    |   movel([0.169835, -1.400800, -2.552340, -0.759249, 1.570796, 1.740631],accel_mss,speed_ms,0,blend_radius_m)
    |   movel([0.168721, -1.399189, -2.553525, -0.759676, 1.570796, 1.739517],accel_mss,speed_ms,0,blend_radius_m)
    |   movel([0.167272, -1.397802, -2.554541, -0.760046, 1.570796, 1.738068],accel_mss,speed_ms,0,blend_radius_m)
    |   movel([0.165480, -1.396676, -2.555365, -0.760348, 1.570796, 1.736276],accel_mss,speed_ms,0,blend_radius_m)
    |   movel([0.163342, -1.395840, -2.555975, -0.760574, 1.570796, 1.734139],accel_mss,speed_ms,0,blend_radius_m)
    |   # Splitting Linear movement in 6 (instruction 331: MoveL 300)
    |   movel([0.161964, -1.395450, -2.556260, -0.760680, 1.570796, 1.732760],accel_mss,speed_ms,0,blend_radius_m)
    |   movel([0.160583, -1.395061, -2.556543, -0.760786, 1.570796, 1.731379],accel_mss,speed_ms,0,blend_radius_m)
    |   movel([0.159200, -1.394674, -2.556824, -0.760891, 1.570796, 1.729996],accel_mss,speed_ms,0,blend_radius_m)
    |   movel([0.157815, -1.394290, -2.557104, -0.760996, 1.570796, 1.728611],accel_mss,speed_ms,0,blend_radius_m)
    |   movel([0.156427, -1.393907, -2.557382, -0.761100, 1.570796, 1.727224],accel_mss,speed_ms,0,blend_radius_m)
    |   movel([0.155038, -1.393527, -2.557658, -0.761204, 1.570796, 1.725834],accel_mss,speed_ms,0,blend_radius_m)
    |   # Splitting Linear movement in 18 (instruction 332: MoveL 301)
    |   movel([0.153192, -1.393056, -2.557999, -0.761333, 1.570796, 1.723988],accel_mss,speed_ms,0,blend_radius_m)
    |   movel([0.151342, -1.392590, -2.558337, -0.761462, 1.570796, 1.722138],accel_mss,speed_ms,0,blend_radius_m)
    |   movel([0.149489, -1.392127, -2.558673, -0.761589, 1.570796, 1.720285],accel_mss,speed_ms,0,blend_radius_m)
    |   movel([0.147632, -1.391668, -2.559005, -0.761716, 1.570796, 1.718428],accel_mss,speed_ms,0,blend_radius_m)
    |   movel([0.145771, -1.391213, -2.559334, -0.761842, 1.570796, 1.716568],accel_mss,speed_ms,0,blend_radius_m)
    |   movel([0.143907, -1.390762, -2.559660, -0.761968, 1.570796, 1.714704],accel_mss,speed_ms,0,blend_radius_m)
    |   movel([0.142040, -1.390314, -2.559982, -0.762092, 1.570796, 1.712836],accel_mss,speed_ms,0,blend_radius_m)
    |   movel([0.140169, -1.389871, -2.560302, -0.762216, 1.570796, 1.710965],accel_mss,speed_ms,0,blend_radius_m)
    |   movel([0.138294, -1.389431, -2.560619, -0.762339, 1.570796, 1.709091],accel_mss,speed_ms,0,blend_radius_m)
    |   movel([0.136416, -1.388995, -2.560933, -0.762461, 1.570796, 1.707213],accel_mss,speed_ms,0,blend_radius_m)
    |   movel([0.134535, -1.388563, -2.561243, -0.762583, 1.570796, 1.705331],accel_mss,speed_ms,0,blend_radius_m)
    |   movel([0.132650, -1.388135, -2.561550, -0.762703, 1.570796, 1.703446],accel_mss,speed_ms,0,blend_radius_m)
    |   movel([0.130761, -1.387711, -2.561855, -0.762823, 1.570796, 1.701558],accel_mss,speed_ms,0,blend_radius_m)
    |   movel([0.128869, -1.387291, -2.562156, -0.762942, 1.570796, 1.699666],accel_mss,speed_ms,0,blend_radius_m)
    |   movel([0.126974, -1.386875, -2.562454, -0.763060, 1.570796, 1.697770],accel_mss,speed_ms,0,blend_radius_m)
    |   movel([0.125075, -1.386463, -2.562749, -0.763177, 1.570796, 1.695872],accel_mss,speed_ms,0,blend_radius_m)
    |   movel([0.123173, -1.386055, -2.563041, -0.763293, 1.570796, 1.693969],accel_mss,speed_ms,0,blend_radius_m)
    |   movel([0.121267, -1.385651, -2.563330, -0.763408, 1.570796, 1.692064],accel_mss,speed_ms,0,blend_radius_m)
    |   movel([0.119799, -1.385268, -2.563603, -0.763517, 1.570796, 1.690595],accel_mss,speed_ms,0,blend_radius_m)
    |   movel([0.119411, -1.385044, -2.563763, -0.763581, 1.570796, 1.690207],accel_mss,speed_ms,0,blend_radius_m)
    |   movel([0.119247, -1.384741, -2.563979, -0.763668, 1.570796, 1.690044],accel_mss,speed_ms,0,blend_radius_m)
    |   movel([0.119299, -1.384311, -2.564286, -0.763792, 1.570796, 1.690095],accel_mss,speed_ms,0,blend_radius_m)
    |   movel([0.119560, -1.383712, -2.564713, -0.763964, 1.570796, 1.690357],accel_mss,speed_ms,0,blend_radius_m)
    |   movel([0.120675, -1.381827, -2.566051, -0.764510, 1.570796, 1.691472],accel_mss,speed_ms,0,blend_radius_m)
    |   movel([0.122734, -1.382263, -2.565743, -0.764384, 1.570796, 1.693530],accel_mss,speed_ms,0,blend_radius_m)
    |   speed_ms = 0.005
    |   # Splitting Linear movement in 4 (instruction 341: MoveL 309)
    |   movel([0.122734, -1.380104, -2.564747, -0.767538, 1.570796, 1.693530],accel_mss,speed_ms,0,blend_radius_m)
    |   movel([0.122734, -1.377955, -2.563748, -0.770686, 1.570796, 1.693530],accel_mss,speed_ms,0,blend_radius_m)
    |   movel([0.122734, -1.375816, -2.562745, -0.773828, 1.570796, 1.693530],accel_mss,speed_ms,0,blend_radius_m)
    |   movel([0.122734, -1.373687, -2.561739, -0.776963, 1.570796, 1.693530],accel_mss,speed_ms,0,blend_radius_m)
    |   speed_ms = 0.040
    |   # Splitting Linear movement in 18 (instruction 343: MoveL 310)
    |   movel([0.125073, -1.372444, -2.562608, -0.777337, 1.570796, 1.695869],accel_mss,speed_ms,0,blend_radius_m)
    |   movel([0.127416, -1.371202, -2.563475, -0.777712, 1.570796, 1.698212],accel_mss,speed_ms,0,blend_radius_m)
    |   movel([0.129763, -1.369961, -2.564339, -0.778089, 1.570796, 1.700560],accel_mss,speed_ms,0,blend_radius_m)
    |   movel([0.132116, -1.368721, -2.565200, -0.778468, 1.570796, 1.702912],accel_mss,speed_ms,0,blend_radius_m)
    |   movel([0.134472, -1.367482, -2.566059, -0.778849, 1.570796, 1.705269],accel_mss,speed_ms,0,blend_radius_m)
    |   movel([0.136834, -1.366243, -2.566914, -0.779232, 1.570796, 1.707630],accel_mss,speed_ms,0,blend_radius_m)
    |   movel([0.139200, -1.365006, -2.567767, -0.779616, 1.570796, 1.709996],accel_mss,speed_ms,0,blend_radius_m)
    |   movel([0.141570, -1.363769, -2.568617, -0.780003, 1.570796, 1.712366],accel_mss,speed_ms,0,blend_radius_m)
    |   movel([0.143945, -1.362533, -2.569465, -0.780391, 1.570796, 1.714741],accel_mss,speed_ms,0,blend_radius_m)
    |   movel([0.146324, -1.361298, -2.570309, -0.780781, 1.570796, 1.717121],accel_mss,speed_ms,0,blend_radius_m)
    |   movel([0.148708, -1.360065, -2.571151, -0.781173, 1.570796, 1.719505],accel_mss,speed_ms,0,blend_radius_m)
    |   movel([0.151097, -1.358832, -2.571990, -0.781567, 1.570796, 1.721893],accel_mss,speed_ms,0,blend_radius_m)
    |   movel([0.153490, -1.357600, -2.572826, -0.781962, 1.570796, 1.724286],accel_mss,speed_ms,0,blend_radius_m)
    |   movel([0.155887, -1.356370, -2.573660, -0.782360, 1.570796, 1.726684],accel_mss,speed_ms,0,blend_radius_m)
    |   movel([0.158289, -1.355140, -2.574490, -0.782759, 1.570796, 1.729086],accel_mss,speed_ms,0,blend_radius_m)
    |   movel([0.160696, -1.353911, -2.575318, -0.783159, 1.570796, 1.731492],accel_mss,speed_ms,0,blend_radius_m)
    |   movel([0.163106, -1.352684, -2.576143, -0.783562, 1.570796, 1.733903],accel_mss,speed_ms,0,blend_radius_m)
    |   movel([0.165522, -1.351458, -2.576965, -0.783966, 1.570796, 1.736318],accel_mss,speed_ms,0,blend_radius_m)
    |   speed_ms = 0.005
    |   # Splitting Linear movement in 6 (instruction 345: MoveL 311)
    |   movel([0.165522, -1.352900, -2.577653, -0.781836, 1.570796, 1.736318],accel_mss,speed_ms,0,blend_radius_m)
    |   movel([0.165522, -1.354347, -2.578339, -0.779703, 1.570796, 1.736318],accel_mss,speed_ms,0,blend_radius_m)
    |   movel([0.165522, -1.355799, -2.579023, -0.777567, 1.570796, 1.736318],accel_mss,speed_ms,0,blend_radius_m)
    |   movel([0.165522, -1.357255, -2.579705, -0.775428, 1.570796, 1.736318],accel_mss,speed_ms,0,blend_radius_m)
    |   movel([0.165522, -1.358716, -2.580386, -0.773287, 1.570796, 1.736318],accel_mss,speed_ms,0,blend_radius_m)
    |   movel([0.165522, -1.360182, -2.581065, -0.771142, 1.570796, 1.736318],accel_mss,speed_ms,0,blend_radius_m)
    |   speed_ms = 0.035
    |   movel([0.167244, -1.360441, -2.580889, -0.771058, 1.570796, 1.738040],accel_mss,speed_ms,0,blend_radius_m)
    |   movel([0.168585, -1.360439, -2.580891, -0.771059, 1.570796, 1.739382],accel_mss,speed_ms,0,blend_radius_m)
    |   movel([0.169955, -1.360315, -2.580975, -0.771099, 1.570796, 1.740751],accel_mss,speed_ms,0,blend_radius_m)
    |   movel([0.171344, -1.360075, -2.581138, -0.771176, 1.570796, 1.742141],accel_mss,speed_ms,0,blend_radius_m)
    |   movel([0.172746, -1.359724, -2.581376, -0.771289, 1.570796, 1.743542],accel_mss,speed_ms,0,blend_radius_m)
    |   movel([0.174155, -1.359265, -2.581687, -0.771437, 1.570796, 1.744951],accel_mss,speed_ms,0,blend_radius_m)
    |   movel([0.176950, -1.358045, -2.582512, -0.771832, 1.570796, 1.747746],accel_mss,speed_ms,0,blend_radius_m)
    |   movel([0.178323, -1.357292, -2.583020, -0.772077, 1.570796, 1.749120],accel_mss,speed_ms,0,blend_radius_m)
    |   movel([0.180981, -1.355525, -2.584210, -0.772655, 1.570796, 1.751777],accel_mss,speed_ms,0,blend_radius_m)
    |   movel([0.182252, -1.354517, -2.584886, -0.772986, 1.570796, 1.753048],accel_mss,speed_ms,0,blend_radius_m)
    |   movel([0.184624, -1.352283, -2.586380, -0.773726, 1.570796, 1.755420],accel_mss,speed_ms,0,blend_radius_m)
    |   movel([0.185715, -1.351062, -2.587194, -0.774133, 1.570796, 1.756511],accel_mss,speed_ms,0,blend_radius_m)
    |   movel([0.186729, -1.349776, -2.588049, -0.774564, 1.570796, 1.757525],accel_mss,speed_ms,0,blend_radius_m)
    |   movel([0.187656, -1.348435, -2.588938, -0.775016, 1.570796, 1.758453],accel_mss,speed_ms,0,blend_radius_m)
    |   movel([0.188445, -1.347113, -2.589812, -0.775464, 1.570796, 1.759241],accel_mss,speed_ms,0,blend_radius_m)
    |   movel([0.189111, -1.345791, -2.590684, -0.775914, 1.570796, 1.759907],accel_mss,speed_ms,0,blend_radius_m)
    |   movel([0.190069, -1.343183, -2.592397, -0.776810, 1.570796, 1.760866],accel_mss,speed_ms,0,blend_radius_m)
    |   movel([0.190366, -1.341908, -2.593230, -0.777251, 1.570796, 1.761162],accel_mss,speed_ms,0,blend_radius_m)
    |   movel([0.190585, -1.339465, -2.594822, -0.778102, 1.570796, 1.761381],accel_mss,speed_ms,0,blend_radius_m)
    |   movel([0.190509, -1.338309, -2.595572, -0.778508, 1.570796, 1.761306],accel_mss,speed_ms,0,blend_radius_m)
    |   movel([0.189997, -1.336168, -2.596957, -0.779265, 1.570796, 1.760793],accel_mss,speed_ms,0,blend_radius_m)
    |   movel([0.189557, -1.335195, -2.597584, -0.779610, 1.570796, 1.760353],accel_mss,speed_ms,0,blend_radius_m)
    |   movel([0.188317, -1.333493, -2.598678, -0.780218, 1.570796, 1.759113],accel_mss,speed_ms,0,blend_radius_m)
    |   movel([0.187516, -1.332779, -2.599136, -0.780474, 1.570796, 1.758312],accel_mss,speed_ms,0,blend_radius_m)
    |   movel([0.186599, -1.332164, -2.599530, -0.780696, 1.570796, 1.757395],accel_mss,speed_ms,0,blend_radius_m)
    |   movel([0.185562, -1.331657, -2.599854, -0.780878, 1.570796, 1.756358],accel_mss,speed_ms,0,blend_radius_m)
    |   movel([0.183890, -1.331154, -2.600175, -0.781060, 1.570796, 1.754686],accel_mss,speed_ms,0,blend_radius_m)
    |   movel([0.183257, -1.331163, -2.600169, -0.781057, 1.570796, 1.754053],accel_mss,speed_ms,0,blend_radius_m)
    |   movel([0.182728, -1.331365, -2.600040, -0.780983, 1.570796, 1.753524],accel_mss,speed_ms,0,blend_radius_m)
    |   movel([0.182274, -1.331780, -2.599775, -0.780834, 1.570796, 1.753070],accel_mss,speed_ms,0,blend_radius_m)
    |   movel([0.181874, -1.332416, -2.599368, -0.780605, 1.570796, 1.752671],accel_mss,speed_ms,0,blend_radius_m)
    |   movel([0.181131, -1.334429, -2.598077, -0.779883, 1.570796, 1.751927],accel_mss,speed_ms,0,blend_radius_m)
    |   movel([0.182746, -1.334997, -2.597711, -0.779681, 1.570796, 1.753542],accel_mss,speed_ms,0,blend_radius_m)
    |   movel([0.184246, -1.335833, -2.597173, -0.779383, 1.570796, 1.755043],accel_mss,speed_ms,0,blend_radius_m)
    |   movel([0.185396, -1.336953, -2.596450, -0.778986, 1.570796, 1.756192],accel_mss,speed_ms,0,blend_radius_m)
    |   movel([0.186193, -1.338317, -2.595567, -0.778505, 1.570796, 1.756989],accel_mss,speed_ms,0,blend_radius_m)
    |   movel([0.186629, -1.339885, -2.594549, -0.777955, 1.570796, 1.757425],accel_mss,speed_ms,0,blend_radius_m)
    |   movel([0.186702, -1.341619, -2.593419, -0.777351, 1.570796, 1.757498],accel_mss,speed_ms,0,blend_radius_m)
    |   movel([0.186412, -1.343480, -2.592202, -0.776707, 1.570796, 1.757208],accel_mss,speed_ms,0,blend_radius_m)
    |   movel([0.185753, -1.345430, -2.590921, -0.776037, 1.570796, 1.756550],accel_mss,speed_ms,0,blend_radius_m)
    |   movel([0.184722, -1.347430, -2.589603, -0.775356, 1.570796, 1.755519],accel_mss,speed_ms,0,blend_radius_m)
    |   movel([0.183346, -1.349406, -2.588295, -0.774688, 1.570796, 1.754142],accel_mss,speed_ms,0,blend_radius_m)
    |   movel([0.181729, -1.351210, -2.587095, -0.774083, 1.570796, 1.752525],accel_mss,speed_ms,0,blend_radius_m)
    |   movel([0.179917, -1.352823, -2.586020, -0.773546, 1.570796, 1.750714],accel_mss,speed_ms,0,blend_radius_m)
    |   movel([0.177958, -1.354214, -2.585089, -0.773086, 1.570796, 1.748754],accel_mss,speed_ms,0,blend_radius_m)
    |   movel([0.175895, -1.355355, -2.584323, -0.772710, 1.570796, 1.746691],accel_mss,speed_ms,0,blend_radius_m)
    |   movel([0.173775, -1.356220, -2.583742, -0.772427, 1.570796, 1.744572],accel_mss,speed_ms,0,blend_radius_m)
    |   movel([0.171644, -1.356782, -2.583364, -0.772243, 1.570796, 1.742441],accel_mss,speed_ms,0,blend_radius_m)
    |   movel([0.169547, -1.357011, -2.583210, -0.772169, 1.570796, 1.740343],accel_mss,speed_ms,0,blend_radius_m)
    |   movel([0.167897, -1.357114, -2.583140, -0.772135, 1.570796, 1.738693],accel_mss,speed_ms,0,blend_radius_m)
    |   movel([0.167339, -1.357255, -2.583045, -0.772089, 1.570796, 1.738135],accel_mss,speed_ms,0,blend_radius_m)
    |   movel([0.166903, -1.357499, -2.582881, -0.772010, 1.570796, 1.737699],accel_mss,speed_ms,0,blend_radius_m)
    |   movel([0.166548, -1.357878, -2.582625, -0.771886, 1.570796, 1.737344],accel_mss,speed_ms,0,blend_radius_m)
    |   movel([0.166226, -1.358432, -2.582251, -0.771707, 1.570796, 1.737022],accel_mss,speed_ms,0,blend_radius_m)
    |   movel([0.165522, -1.360182, -2.581065, -0.771142, 1.570796, 1.736318],accel_mss,speed_ms,0,blend_radius_m)
    |   movel([0.167244, -1.360441, -2.580889, -0.771058, 1.570796, 1.738040],accel_mss,speed_ms,0,blend_radius_m)
    |   movel([0.167727, -1.360442, -2.580889, -0.771058, 1.570796, 1.738523],accel_mss,speed_ms,0,blend_radius_m)
    |   speed_ms = 0.005
    |   # Splitting Linear movement in 6 (instruction 405: MoveL 369)
    |   movel([0.167727, -1.358977, -2.580210, -0.773202, 1.570796, 1.738523],accel_mss,speed_ms,0,blend_radius_m)
    |   movel([0.167727, -1.357516, -2.579529, -0.775344, 1.570796, 1.738523],accel_mss,speed_ms,0,blend_radius_m)
    |   movel([0.167727, -1.356060, -2.578847, -0.777482, 1.570796, 1.738523],accel_mss,speed_ms,0,blend_radius_m)
    |   movel([0.167727, -1.354609, -2.578163, -0.779618, 1.570796, 1.738523],accel_mss,speed_ms,0,blend_radius_m)
    |   movel([0.167727, -1.353162, -2.577477, -0.781750, 1.570796, 1.738523],accel_mss,speed_ms,0,blend_radius_m)
    |   movel([0.167727, -1.351720, -2.576790, -0.783879, 1.570796, 1.738523],accel_mss,speed_ms,0,blend_radius_m)
    |   speed_ms = 0.040
    |   # Splitting Linear movement in 6 (instruction 407: MoveL 370)
    |   movel([0.165743, -1.351292, -2.577077, -0.784021, 1.570796, 1.736539],accel_mss,speed_ms,0,blend_radius_m)
    |   movel([0.163755, -1.350868, -2.577360, -0.784161, 1.570796, 1.734551],accel_mss,speed_ms,0,blend_radius_m)
    |   movel([0.161764, -1.350449, -2.577640, -0.784300, 1.570796, 1.732560],accel_mss,speed_ms,0,blend_radius_m)
    |   movel([0.159768, -1.350034, -2.577917, -0.784438, 1.570796, 1.730565],accel_mss,speed_ms,0,blend_radius_m)
    |   movel([0.157769, -1.349624, -2.578191, -0.784574, 1.570796, 1.728566],accel_mss,speed_ms,0,blend_radius_m)
    |   movel([0.155767, -1.349218, -2.578462, -0.784709, 1.570796, 1.726563],accel_mss,speed_ms,0,blend_radius_m)
    |   speed_ms = 0.005
    |   # Splitting Linear movement in 6 (instruction 409: MoveL 371)
    |   movel([0.155767, -1.350663, -2.579151, -0.782575, 1.570796, 1.726563],accel_mss,speed_ms,0,blend_radius_m)
    |   movel([0.155767, -1.352112, -2.579838, -0.780439, 1.570796, 1.726563],accel_mss,speed_ms,0,blend_radius_m)
    |   movel([0.155767, -1.353567, -2.580524, -0.778299, 1.570796, 1.726563],accel_mss,speed_ms,0,blend_radius_m)
    |   movel([0.155767, -1.355025, -2.581208, -0.776156, 1.570796, 1.726563],accel_mss,speed_ms,0,blend_radius_m)
    |   movel([0.155767, -1.356489, -2.581891, -0.774010, 1.570796, 1.726563],accel_mss,speed_ms,0,blend_radius_m)
    |   movel([0.155767, -1.357957, -2.582571, -0.771861, 1.570796, 1.726563],accel_mss,speed_ms,0,blend_radius_m)
    |   speed_ms = 0.035
    |   movel([0.157355, -1.355183, -2.584439, -0.772767, 1.570796, 1.728151],accel_mss,speed_ms,0,blend_radius_m)
    |   movel([0.158736, -1.352483, -2.586247, -0.773659, 1.570796, 1.729532],accel_mss,speed_ms,0,blend_radius_m)
    |   movel([0.159906, -1.349859, -2.587994, -0.774536, 1.570796, 1.730702],accel_mss,speed_ms,0,blend_radius_m)
    |   movel([0.160863, -1.347310, -2.589682, -0.775397, 1.570796, 1.731660],accel_mss,speed_ms,0,blend_radius_m)
    |   movel([0.161608, -1.344839, -2.591310, -0.776240, 1.570796, 1.732405],accel_mss,speed_ms,0,blend_radius_m)
    |   movel([0.162137, -1.342441, -2.592882, -0.777066, 1.570796, 1.732933],accel_mss,speed_ms,0,blend_radius_m)
    |   movel([0.162447, -1.340121, -2.594395, -0.777873, 1.570796, 1.733244],accel_mss,speed_ms,0,blend_radius_m)
    |   movel([0.162537, -1.337882, -2.595848, -0.778658, 1.570796, 1.733334],accel_mss,speed_ms,0,blend_radius_m)
    |   movel([0.162403, -1.335721, -2.597245, -0.779423, 1.570796, 1.733200],accel_mss,speed_ms,0,blend_radius_m)
    |   movel([0.162046, -1.333638, -2.598585, -0.780166, 1.570796, 1.732842],accel_mss,speed_ms,0,blend_radius_m)
    |   movel([0.161461, -1.331638, -2.599866, -0.780885, 1.570796, 1.732257],accel_mss,speed_ms,0,blend_radius_m)
    |   movel([0.160647, -1.329720, -2.601089, -0.781580, 1.570796, 1.731443],accel_mss,speed_ms,0,blend_radius_m)
    |   movel([0.159603, -1.327887, -2.602254, -0.782248, 1.570796, 1.730399],accel_mss,speed_ms,0,blend_radius_m)
    |   movel([0.158326, -1.326137, -2.603362, -0.782890, 1.570796, 1.729123],accel_mss,speed_ms,0,blend_radius_m)
    |   movel([0.156817, -1.324475, -2.604410, -0.783504, 1.570796, 1.727613],accel_mss,speed_ms,0,blend_radius_m)
    |   movel([0.155070, -1.322901, -2.605399, -0.784089, 1.570796, 1.725866],accel_mss,speed_ms,0,blend_radius_m)
    |   movel([0.156422, -1.321887, -2.606034, -0.784467, 1.570796, 1.727219],accel_mss,speed_ms,0,blend_radius_m)
    |   movel([0.158344, -1.320258, -2.607053, -0.785078, 1.570796, 1.729140],accel_mss,speed_ms,0,blend_radius_m)
    |   movel([0.160279, -1.321620, -2.606202, -0.784567, 1.570796, 1.731076],accel_mss,speed_ms,0,blend_radius_m)
    |   movel([0.161946, -1.323240, -2.605186, -0.783963, 1.570796, 1.732742],accel_mss,speed_ms,0,blend_radius_m)
    |   movel([0.163339, -1.325091, -2.604022, -0.783276, 1.570796, 1.734136],accel_mss,speed_ms,0,blend_radius_m)
    |   movel([0.164467, -1.327149, -2.602721, -0.782518, 1.570796, 1.735263],accel_mss,speed_ms,0,blend_radius_m)
    |   movel([0.165329, -1.329385, -2.601302, -0.781701, 1.570796, 1.736126],accel_mss,speed_ms,0,blend_radius_m)
    |   movel([0.165930, -1.331777, -2.599777, -0.780835, 1.570796, 1.736726],accel_mss,speed_ms,0,blend_radius_m)
    |   movel([0.166274, -1.334295, -2.598163, -0.779931, 1.570796, 1.737070],accel_mss,speed_ms,0,blend_radius_m)
    |   movel([0.166364, -1.336915, -2.596474, -0.779000, 1.570796, 1.737160],accel_mss,speed_ms,0,blend_radius_m)
    |   movel([0.166202, -1.339614, -2.594725, -0.778050, 1.570796, 1.736998],accel_mss,speed_ms,0,blend_radius_m)
    |   movel([0.165795, -1.342364, -2.592932, -0.777093, 1.570796, 1.736591],accel_mss,speed_ms,0,blend_radius_m)
    |   movel([0.165144, -1.345146, -2.591108, -0.776135, 1.570796, 1.735940],accel_mss,speed_ms,0,blend_radius_m)
    |   movel([0.164254, -1.347930, -2.589272, -0.775187, 1.570796, 1.735050],accel_mss,speed_ms,0,blend_radius_m)
    |   movel([0.163128, -1.350701, -2.587435, -0.774254, 1.570796, 1.733924],accel_mss,speed_ms,0,blend_radius_m)
    |   movel([0.161769, -1.353431, -2.585613, -0.773345, 1.570796, 1.732566],accel_mss,speed_ms,0,blend_radius_m)
    |   movel([0.160179, -1.356100, -2.583823, -0.772466, 1.570796, 1.730976],accel_mss,speed_ms,0,blend_radius_m)
    |   movel([0.158366, -1.358687, -2.582078, -0.771624, 1.570796, 1.729162],accel_mss,speed_ms,0,blend_radius_m)
    |   movel([0.155767, -1.357957, -2.582571, -0.771861, 1.570796, 1.726563],accel_mss,speed_ms,0,blend_radius_m)
    |   movel([0.157104, -1.355619, -2.584147, -0.772624, 1.570796, 1.727901],accel_mss,speed_ms,0,blend_radius_m)
    |   speed_ms = 0.005
    |   # Splitting Linear movement in 6 (instruction 448: MoveL 408)
    |   movel([0.157104, -1.354148, -2.583464, -0.774777, 1.570796, 1.727901],accel_mss,speed_ms,0,blend_radius_m)
    |   movel([0.157104, -1.352682, -2.582780, -0.776927, 1.570796, 1.727901],accel_mss,speed_ms,0,blend_radius_m)
    |   movel([0.157104, -1.351221, -2.582094, -0.779075, 1.570796, 1.727901],accel_mss,speed_ms,0,blend_radius_m)
    |   movel([0.157104, -1.349764, -2.581406, -0.781219, 1.570796, 1.727901],accel_mss,speed_ms,0,blend_radius_m)
    |   movel([0.157104, -1.348312, -2.580717, -0.783360, 1.570796, 1.727901],accel_mss,speed_ms,0,blend_radius_m)
    |   movel([0.157104, -1.346865, -2.580026, -0.785498, 1.570796, 1.727901],accel_mss,speed_ms,0,blend_radius_m)
    |   speed_ms = 0.040
    |   # Splitting Linear movement in 6 (instruction 450: MoveL 409)
    |   movel([0.154683, -1.347404, -2.579668, -0.785317, 1.570796, 1.725480],accel_mss,speed_ms,0,blend_radius_m)
    |   movel([0.152263, -1.347947, -2.579307, -0.785134, 1.570796, 1.723059],accel_mss,speed_ms,0,blend_radius_m)
    |   movel([0.149843, -1.348495, -2.578943, -0.784951, 1.570796, 1.720639],accel_mss,speed_ms,0,blend_radius_m)
    |   movel([0.147424, -1.349048, -2.578575, -0.784766, 1.570796, 1.718220],accel_mss,speed_ms,0,blend_radius_m)
    |   movel([0.145005, -1.349604, -2.578204, -0.784581, 1.570796, 1.715801],accel_mss,speed_ms,0,blend_radius_m)
    |   movel([0.142587, -1.350165, -2.577830, -0.784394, 1.570796, 1.713383],accel_mss,speed_ms,0,blend_radius_m)
    |   speed_ms = 0.005
    |   # Splitting Linear movement in 6 (instruction 452: MoveL 410)
    |   movel([0.142587, -1.351609, -2.578518, -0.782262, 1.570796, 1.713383],accel_mss,speed_ms,0,blend_radius_m)
    |   movel([0.142587, -1.353057, -2.579205, -0.780127, 1.570796, 1.713383],accel_mss,speed_ms,0,blend_radius_m)
    |   movel([0.142587, -1.354510, -2.579890, -0.777989, 1.570796, 1.713383],accel_mss,speed_ms,0,blend_radius_m)
    |   movel([0.142587, -1.355968, -2.580574, -0.775847, 1.570796, 1.713383],accel_mss,speed_ms,0,blend_radius_m)
    |   movel([0.142587, -1.357430, -2.581256, -0.773703, 1.570796, 1.713383],accel_mss,speed_ms,0,blend_radius_m)
    |   movel([0.142587, -1.358897, -2.581936, -0.771556, 1.570796, 1.713383],accel_mss,speed_ms,0,blend_radius_m)
    |   speed_ms = 0.035
    |   movel([0.144618, -1.357853, -2.582642, -0.771895, 1.570796, 1.715414],accel_mss,speed_ms,0,blend_radius_m)
    |   movel([0.145265, -1.357609, -2.582806, -0.771974, 1.570796, 1.716061],accel_mss,speed_ms,0,blend_radius_m)
    |   movel([0.145714, -1.357563, -2.582837, -0.771989, 1.570796, 1.716510],accel_mss,speed_ms,0,blend_radius_m)
    |   movel([0.146013, -1.357716, -2.582734, -0.771939, 1.570796, 1.716810],accel_mss,speed_ms,0,blend_radius_m)
    |   movel([0.146199, -1.358079, -2.582489, -0.771821, 1.570796, 1.716996],accel_mss,speed_ms,0,blend_radius_m)
    |   movel([0.146391, -1.359451, -2.581561, -0.771377, 1.570796, 1.717188],accel_mss,speed_ms,0,blend_radius_m)
    |   movel([0.146678, -1.361399, -2.580239, -0.770751, 1.570796, 1.717475],accel_mss,speed_ms,0,blend_radius_m)
    |   movel([0.147186, -1.363219, -2.578999, -0.770171, 1.570796, 1.717982],accel_mss,speed_ms,0,blend_radius_m)
    |   movel([0.147904, -1.364903, -2.577847, -0.769639, 1.570796, 1.718700],accel_mss,speed_ms,0,blend_radius_m)
    |   movel([0.148823, -1.366444, -2.576790, -0.769155, 1.570796, 1.719620],accel_mss,speed_ms,0,blend_radius_m)
    |   movel([0.149928, -1.367838, -2.575830, -0.768720, 1.570796, 1.720724],accel_mss,speed_ms,0,blend_radius_m)
    |   movel([0.151213, -1.369078, -2.574975, -0.768336, 1.570796, 1.722009],accel_mss,speed_ms,0,blend_radius_m)
    |   movel([0.152668, -1.370158, -2.574228, -0.768003, 1.570796, 1.723464],accel_mss,speed_ms,0,blend_radius_m)
    |   movel([0.154279, -1.371073, -2.573594, -0.767722, 1.570796, 1.725075],accel_mss,speed_ms,0,blend_radius_m)
    |   movel([0.156039, -1.371815, -2.573079, -0.767495, 1.570796, 1.726835],accel_mss,speed_ms,0,blend_radius_m)
    |   movel([0.157942, -1.372376, -2.572689, -0.767324, 1.570796, 1.728738],accel_mss,speed_ms,0,blend_radius_m)
    |   movel([0.159972, -1.372753, -2.572427, -0.767209, 1.570796, 1.730769],accel_mss,speed_ms,0,blend_radius_m)
    |   movel([0.162127, -1.372933, -2.572301, -0.767155, 1.570796, 1.732924],accel_mss,speed_ms,0,blend_radius_m)
    |   movel([0.164395, -1.372914, -2.572314, -0.767160, 1.570796, 1.735192],accel_mss,speed_ms,0,blend_radius_m)
    |   movel([0.166771, -1.372686, -2.572473, -0.767230, 1.570796, 1.737567],accel_mss,speed_ms,0,blend_radius_m)
    |   movel([0.169243, -1.372241, -2.572783, -0.767365, 1.570796, 1.740039],accel_mss,speed_ms,0,blend_radius_m)
    |   movel([0.171807, -1.371570, -2.573249, -0.767570, 1.570796, 1.742603],accel_mss,speed_ms,0,blend_radius_m)
    |   movel([0.174557, -1.370640, -2.573894, -0.767855, 1.570796, 1.745353],accel_mss,speed_ms,0,blend_radius_m)
    |   movel([0.177244, -1.369534, -2.574660, -0.768195, 1.570796, 1.748040],accel_mss,speed_ms,0,blend_radius_m)
    |   movel([0.179860, -1.368264, -2.575537, -0.768588, 1.570796, 1.750657],accel_mss,speed_ms,0,blend_radius_m)
    |   movel([0.182392, -1.366838, -2.576519, -0.769032, 1.570796, 1.753189],accel_mss,speed_ms,0,blend_radius_m)
    |   movel([0.184834, -1.365264, -2.577600, -0.769525, 1.570796, 1.755630],accel_mss,speed_ms,0,blend_radius_m)
    |   movel([0.187171, -1.363557, -2.578768, -0.770064, 1.570796, 1.757967],accel_mss,speed_ms,0,blend_radius_m)
    |   movel([0.189395, -1.361724, -2.580018, -0.770647, 1.570796, 1.760191],accel_mss,speed_ms,0,blend_radius_m)
    |   movel([0.191497, -1.359772, -2.581343, -0.771274, 1.570796, 1.762293],accel_mss,speed_ms,0,blend_radius_m)
    |   movel([0.193462, -1.357715, -2.582735, -0.771939, 1.570796, 1.764258],accel_mss,speed_ms,0,blend_radius_m)
    |   movel([0.195284, -1.355561, -2.584185, -0.772643, 1.570796, 1.766080],accel_mss,speed_ms,0,blend_radius_m)
    |   movel([0.196947, -1.353323, -2.585686, -0.773381, 1.570796, 1.767743],accel_mss,speed_ms,0,blend_radius_m)
    |   movel([0.198441, -1.351008, -2.587230, -0.774151, 1.570796, 1.769238],accel_mss,speed_ms,0,blend_radius_m)
    |   movel([0.199751, -1.348631, -2.588808, -0.774950, 1.570796, 1.770547],accel_mss,speed_ms,0,blend_radius_m)
    |   movel([0.200870, -1.346200, -2.590415, -0.775775, 1.570796, 1.771666],accel_mss,speed_ms,0,blend_radius_m)
    |   movel([0.201780, -1.343726, -2.592041, -0.776623, 1.570796, 1.772576],accel_mss,speed_ms,0,blend_radius_m)
    |   movel([0.202469, -1.341224, -2.593677, -0.777488, 1.570796, 1.773266],accel_mss,speed_ms,0,blend_radius_m)
    |   movel([0.202849, -1.339180, -2.595007, -0.778202, 1.570796, 1.773645],accel_mss,speed_ms,0,blend_radius_m)
    |   movel([0.203044, -1.337202, -2.596289, -0.778898, 1.570796, 1.773841],accel_mss,speed_ms,0,blend_radius_m)
    |   movel([0.203058, -1.335296, -2.597519, -0.779574, 1.570796, 1.773854],accel_mss,speed_ms,0,blend_radius_m)
    |   movel([0.202894, -1.333475, -2.598690, -0.780225, 1.570796, 1.773690],accel_mss,speed_ms,0,blend_radius_m)
    |   movel([0.202553, -1.331740, -2.599801, -0.780848, 1.570796, 1.773349],accel_mss,speed_ms,0,blend_radius_m)
    |   movel([0.202041, -1.330104, -2.600845, -0.781440, 1.570796, 1.772837],accel_mss,speed_ms,0,blend_radius_m)
    |   movel([0.201360, -1.328572, -2.601819, -0.781998, 1.570796, 1.772156],accel_mss,speed_ms,0,blend_radius_m)
    |   movel([0.200513, -1.327155, -2.602718, -0.782516, 1.570796, 1.771309],accel_mss,speed_ms,0,blend_radius_m)
    |   movel([0.199505, -1.325856, -2.603539, -0.782994, 1.570796, 1.770301],accel_mss,speed_ms,0,blend_radius_m)
    |   movel([0.198339, -1.324688, -2.604276, -0.783425, 1.570796, 1.769136],accel_mss,speed_ms,0,blend_radius_m)
    |   movel([0.197021, -1.323655, -2.604925, -0.783808, 1.570796, 1.767817],accel_mss,speed_ms,0,blend_radius_m)
    |   movel([0.195555, -1.322767, -2.605483, -0.784139, 1.570796, 1.766352],accel_mss,speed_ms,0,blend_radius_m)
    |   movel([0.193946, -1.322030, -2.605945, -0.784414, 1.570796, 1.764742],accel_mss,speed_ms,0,blend_radius_m)
    |   movel([0.192197, -1.321452, -2.606307, -0.784630, 1.570796, 1.762993],accel_mss,speed_ms,0,blend_radius_m)
    |   movel([0.190314, -1.321041, -2.606564, -0.784784, 1.570796, 1.761110],accel_mss,speed_ms,0,blend_radius_m)
    |   movel([0.188302, -1.320804, -2.606712, -0.784873, 1.570796, 1.759098],accel_mss,speed_ms,0,blend_radius_m)
    |   movel([0.186033, -1.320586, -2.606848, -0.784955, 1.570796, 1.756829],accel_mss,speed_ms,0,blend_radius_m)
    |   movel([0.186699, -1.318620, -2.608073, -0.785696, 1.570796, 1.757495],accel_mss,speed_ms,0,blend_radius_m)
    |   movel([0.187062, -1.317970, -2.608477, -0.785942, 1.570796, 1.757858],accel_mss,speed_ms,0,blend_radius_m)
    |   movel([0.187486, -1.317514, -2.608760, -0.786115, 1.570796, 1.758283],accel_mss,speed_ms,0,blend_radius_m)
    |   movel([0.188004, -1.317220, -2.608942, -0.786227, 1.570796, 1.758800],accel_mss,speed_ms,0,blend_radius_m)
    |   movel([0.188643, -1.317067, -2.609037, -0.786285, 1.570796, 1.759439],accel_mss,speed_ms,0,blend_radius_m)
    |   movel([0.190414, -1.317087, -2.609024, -0.786277, 1.570796, 1.761210],accel_mss,speed_ms,0,blend_radius_m)
    |   movel([0.192754, -1.317403, -2.608829, -0.786157, 1.570796, 1.763550],accel_mss,speed_ms,0,blend_radius_m)
    |   movel([0.194935, -1.317924, -2.608505, -0.785960, 1.570796, 1.765732],accel_mss,speed_ms,0,blend_radius_m)
    |   movel([0.196955, -1.318641, -2.608060, -0.785688, 1.570796, 1.767752],accel_mss,speed_ms,0,blend_radius_m)
    |   movel([0.198804, -1.319549, -2.607495, -0.785345, 1.570796, 1.769600],accel_mss,speed_ms,0,blend_radius_m)
    |   movel([0.200476, -1.320635, -2.606817, -0.784936, 1.570796, 1.771272],accel_mss,speed_ms,0,blend_radius_m)
    |   movel([0.201971, -1.321889, -2.606033, -0.784467, 1.570796, 1.772767],accel_mss,speed_ms,0,blend_radius_m)
    |   movel([0.203277, -1.323305, -2.605146, -0.783939, 1.570796, 1.774073],accel_mss,speed_ms,0,blend_radius_m)
    |   movel([0.204395, -1.324866, -2.604164, -0.783359, 1.570796, 1.775192],accel_mss,speed_ms,0,blend_radius_m)
    |   movel([0.205318, -1.326569, -2.603089, -0.782731, 1.570796, 1.776115],accel_mss,speed_ms,0,blend_radius_m)
    |   movel([0.206044, -1.328398, -2.601930, -0.782061, 1.570796, 1.776841],accel_mss,speed_ms,0,blend_radius_m)
    |   movel([0.206568, -1.330347, -2.600690, -0.781352, 1.570796, 1.777365],accel_mss,speed_ms,0,blend_radius_m)
    |   movel([0.206883, -1.332405, -2.599375, -0.780609, 1.570796, 1.777680],accel_mss,speed_ms,0,blend_radius_m)
    |   movel([0.206991, -1.334560, -2.597992, -0.779836, 1.570796, 1.777788],accel_mss,speed_ms,0,blend_radius_m)
    |   movel([0.206884, -1.336808, -2.596543, -0.779038, 1.570796, 1.777681],accel_mss,speed_ms,0,blend_radius_m)
    |   movel([0.206563, -1.339132, -2.595038, -0.778219, 1.570796, 1.777359],accel_mss,speed_ms,0,blend_radius_m)
    |   movel([0.206022, -1.341527, -2.593479, -0.777383, 1.570796, 1.776818],accel_mss,speed_ms,0,blend_radius_m)
    |   movel([0.205270, -1.343944, -2.591898, -0.776547, 1.570796, 1.776066],accel_mss,speed_ms,0,blend_radius_m)
    |   movel([0.204329, -1.346344, -2.590319, -0.775725, 1.570796, 1.775125],accel_mss,speed_ms,0,blend_radius_m)
    |   movel([0.203206, -1.348721, -2.588749, -0.774919, 1.570796, 1.774003],accel_mss,speed_ms,0,blend_radius_m)
    |   movel([0.201915, -1.351058, -2.587197, -0.774134, 1.570796, 1.772711],accel_mss,speed_ms,0,blend_radius_m)
    |   movel([0.200464, -1.353349, -2.585668, -0.773372, 1.570796, 1.771260],accel_mss,speed_ms,0,blend_radius_m)
    |   movel([0.198867, -1.355583, -2.584170, -0.772635, 1.570796, 1.769664],accel_mss,speed_ms,0,blend_radius_m)
    |   movel([0.197131, -1.357754, -2.582708, -0.771926, 1.570796, 1.767927],accel_mss,speed_ms,0,blend_radius_m)
    |   movel([0.195269, -1.359848, -2.581292, -0.771249, 1.570796, 1.766065],accel_mss,speed_ms,0,blend_radius_m)
    |   movel([0.193289, -1.361860, -2.579925, -0.770604, 1.570796, 1.764085],accel_mss,speed_ms,0,blend_radius_m)
    |   movel([0.191199, -1.363780, -2.578616, -0.769993, 1.570796, 1.761995],accel_mss,speed_ms,0,blend_radius_m)
    |   movel([0.189008, -1.365597, -2.577371, -0.769420, 1.570796, 1.759805],accel_mss,speed_ms,0,blend_radius_m)
    |   movel([0.186730, -1.367307, -2.576197, -0.768886, 1.570796, 1.757527],accel_mss,speed_ms,0,blend_radius_m)
    |   movel([0.184369, -1.368895, -2.575102, -0.768393, 1.570796, 1.755166],accel_mss,speed_ms,0,blend_radius_m)
    |   movel([0.181935, -1.370360, -2.574089, -0.767941, 1.570796, 1.752731],accel_mss,speed_ms,0,blend_radius_m)
    |   movel([0.179436, -1.371687, -2.573168, -0.767534, 1.570796, 1.750233],accel_mss,speed_ms,0,blend_radius_m)
    |   movel([0.176882, -1.372869, -2.572346, -0.767174, 1.570796, 1.747678],accel_mss,speed_ms,0,blend_radius_m)
    |   movel([0.174330, -1.373880, -2.571641, -0.766868, 1.570796, 1.745127],accel_mss,speed_ms,0,blend_radius_m)
    |   movel([0.171808, -1.374709, -2.571062, -0.766618, 1.570796, 1.742604],accel_mss,speed_ms,0,blend_radius_m)
    |   movel([0.169325, -1.375362, -2.570606, -0.766421, 1.570796, 1.740121],accel_mss,speed_ms,0,blend_radius_m)
    |   movel([0.166894, -1.375835, -2.570275, -0.766280, 1.570796, 1.737691],accel_mss,speed_ms,0,blend_radius_m)
    |   movel([0.164518, -1.376135, -2.570065, -0.766190, 1.570796, 1.735315],accel_mss,speed_ms,0,blend_radius_m)
    |   movel([0.162212, -1.376262, -2.569975, -0.766152, 1.570796, 1.733009],accel_mss,speed_ms,0,blend_radius_m)
    |   movel([0.159981, -1.376220, -2.570004, -0.766164, 1.570796, 1.730778],accel_mss,speed_ms,0,blend_radius_m)
    |   movel([0.157837, -1.376006, -2.570155, -0.766228, 1.570796, 1.728633],accel_mss,speed_ms,0,blend_radius_m)
    |   movel([0.155786, -1.375625, -2.570421, -0.766342, 1.570796, 1.726582],accel_mss,speed_ms,0,blend_radius_m)
    |   movel([0.153843, -1.375077, -2.570805, -0.766507, 1.570796, 1.724639],accel_mss,speed_ms,0,blend_radius_m)
    |   movel([0.152016, -1.374360, -2.571306, -0.766723, 1.570796, 1.722813],accel_mss,speed_ms,0,blend_radius_m)
    |   movel([0.150314, -1.373478, -2.571922, -0.766990, 1.570796, 1.721111],accel_mss,speed_ms,0,blend_radius_m)
    |   movel([0.148748, -1.372430, -2.572651, -0.767308, 1.570796, 1.719545],accel_mss,speed_ms,0,blend_radius_m)
    |   movel([0.147329, -1.371214, -2.573496, -0.767679, 1.570796, 1.718125],accel_mss,speed_ms,0,blend_radius_m)
    |   movel([0.146068, -1.369834, -2.574453, -0.768103, 1.570796, 1.716865],accel_mss,speed_ms,0,blend_radius_m)
    |   movel([0.144973, -1.368285, -2.575522, -0.768581, 1.570796, 1.715770],accel_mss,speed_ms,0,blend_radius_m)
    |   movel([0.143879, -1.366214, -2.576948, -0.769227, 1.570796, 1.714675],accel_mss,speed_ms,0,blend_radius_m)
    |   movel([0.143082, -1.363974, -2.578483, -0.769932, 1.570796, 1.713878],accel_mss,speed_ms,0,blend_radius_m)
    |   movel([0.142634, -1.361542, -2.580141, -0.770705, 1.570796, 1.713430],accel_mss,speed_ms,0,blend_radius_m)
    |   movel([0.142587, -1.358897, -2.581936, -0.771556, 1.570796, 1.713383],accel_mss,speed_ms,0,blend_radius_m)
    |   movel([0.144618, -1.357853, -2.582642, -0.771895, 1.570796, 1.715414],accel_mss,speed_ms,0,blend_radius_m)
    |   movel([0.145130, -1.357660, -2.582771, -0.771957, 1.570796, 1.715926],accel_mss,speed_ms,0,blend_radius_m)
    |   speed_ms = 0.005
    |   # Splitting Linear movement in 4 (instruction 570: MoveL 526)
    |   movel([0.145130, -1.355460, -2.581749, -0.775180, 1.570796, 1.715926],accel_mss,speed_ms,0,blend_radius_m)
    |   movel([0.145130, -1.353269, -2.580723, -0.778397, 1.570796, 1.715926],accel_mss,speed_ms,0,blend_radius_m)
    |   movel([0.145130, -1.351089, -2.579694, -0.781606, 1.570796, 1.715926],accel_mss,speed_ms,0,blend_radius_m)
    |   movel([0.145130, -1.348920, -2.578660, -0.784809, 1.570796, 1.715926],accel_mss,speed_ms,0,blend_radius_m)
    |   speed_ms = 0.040
    |   # Splitting Linear movement in 10 (instruction 572: MoveL 527)
    |   movel([0.142834, -1.349486, -2.578283, -0.784620, 1.570796, 1.713630],accel_mss,speed_ms,0,blend_radius_m)
    |   movel([0.140539, -1.350055, -2.577903, -0.784431, 1.570796, 1.711335],accel_mss,speed_ms,0,blend_radius_m)
    |   movel([0.138244, -1.350629, -2.577520, -0.784240, 1.570796, 1.709040],accel_mss,speed_ms,0,blend_radius_m)
    |   movel([0.135951, -1.351206, -2.577134, -0.784049, 1.570796, 1.706747],accel_mss,speed_ms,0,blend_radius_m)
    |   movel([0.133658, -1.351786, -2.576745, -0.783857, 1.570796, 1.704454],accel_mss,speed_ms,0,blend_radius_m)
    |   movel([0.131366, -1.352370, -2.576354, -0.783665, 1.570796, 1.702162],accel_mss,speed_ms,0,blend_radius_m)
    |   movel([0.129075, -1.352958, -2.575959, -0.783472, 1.570796, 1.699871],accel_mss,speed_ms,0,blend_radius_m)
    |   movel([0.126784, -1.353549, -2.575562, -0.783278, 1.570796, 1.697581],accel_mss,speed_ms,0,blend_radius_m)
    |   movel([0.124495, -1.354144, -2.575161, -0.783083, 1.570796, 1.695291],accel_mss,speed_ms,0,blend_radius_m)
    |   movel([0.122207, -1.354743, -2.574758, -0.782888, 1.570796, 1.693003],accel_mss,speed_ms,0,blend_radius_m)
    |   speed_ms = 0.005
    |   # Splitting Linear movement in 4 (instruction 574: MoveL 528)
    |   movel([0.122207, -1.356903, -2.575785, -0.779701, 1.570796, 1.693003],accel_mss,speed_ms,0,blend_radius_m)
    |   movel([0.122207, -1.359074, -2.576808, -0.776507, 1.570796, 1.693003],accel_mss,speed_ms,0,blend_radius_m)
    |   movel([0.122207, -1.361255, -2.577828, -0.773306, 1.570796, 1.693003],accel_mss,speed_ms,0,blend_radius_m)
    |   movel([0.122207, -1.363446, -2.578844, -0.770099, 1.570796, 1.693003],accel_mss,speed_ms,0,blend_radius_m)
    |   speed_ms = 0.035
    |   movel([0.120628, -1.366409, -2.576814, -0.769166, 1.570796, 1.691424],accel_mss,speed_ms,0,blend_radius_m)
    |   movel([0.119214, -1.366251, -2.576922, -0.769215, 1.570796, 1.690010],accel_mss,speed_ms,0,blend_radius_m)
    |   movel([0.117940, -1.365961, -2.577122, -0.769306, 1.570796, 1.688737],accel_mss,speed_ms,0,blend_radius_m)
    |   movel([0.116802, -1.365543, -2.577409, -0.769438, 1.570796, 1.687599],accel_mss,speed_ms,0,blend_radius_m)
    |   movel([0.115794, -1.365001, -2.577780, -0.769608, 1.570796, 1.686590],accel_mss,speed_ms,0,blend_radius_m)
    |   movel([0.114907, -1.364338, -2.578234, -0.769817, 1.570796, 1.685704],accel_mss,speed_ms,0,blend_radius_m)
    |   movel([0.114139, -1.363559, -2.578767, -0.770064, 1.570796, 1.684935],accel_mss,speed_ms,0,blend_radius_m)
    |   movel([0.113482, -1.362670, -2.579373, -0.770346, 1.570796, 1.684278],accel_mss,speed_ms,0,blend_radius_m)
    |   movel([0.112927, -1.361672, -2.580053, -0.770664, 1.570796, 1.683724],accel_mss,speed_ms,0,blend_radius_m)
    |   movel([0.112291, -1.359794, -2.581329, -0.771267, 1.570796, 1.683087],accel_mss,speed_ms,0,blend_radius_m)
    |   movel([0.112068, -1.357735, -2.582721, -0.771933, 1.570796, 1.682864],accel_mss,speed_ms,0,blend_radius_m)
    |   movel([0.112247, -1.355538, -2.584201, -0.772650, 1.570796, 1.683043],accel_mss,speed_ms,0,blend_radius_m)
    |   movel([0.112813, -1.353248, -2.585735, -0.773405, 1.570796, 1.683610],accel_mss,speed_ms,0,blend_radius_m)
    |   movel([0.113756, -1.350904, -2.587299, -0.774186, 1.570796, 1.684553],accel_mss,speed_ms,0,blend_radius_m)
    |   movel([0.115059, -1.348556, -2.588858, -0.774975, 1.570796, 1.685855],accel_mss,speed_ms,0,blend_radius_m)
    |   movel([0.116712, -1.346243, -2.590386, -0.775760, 1.570796, 1.687508],accel_mss,speed_ms,0,blend_radius_m)
    |   movel([0.118694, -1.344015, -2.591851, -0.776523, 1.570796, 1.689491],accel_mss,speed_ms,0,blend_radius_m)
    |   movel([0.120927, -1.341975, -2.593187, -0.777228, 1.570796, 1.691723],accel_mss,speed_ms,0,blend_radius_m)
    |   movel([0.123311, -1.340195, -2.594347, -0.777847, 1.570796, 1.694107],accel_mss,speed_ms,0,blend_radius_m)
    |   movel([0.125806, -1.338693, -2.595323, -0.778373, 1.570796, 1.696602],accel_mss,speed_ms,0,blend_radius_m)
    |   movel([0.128360, -1.337495, -2.596099, -0.778795, 1.570796, 1.699157],accel_mss,speed_ms,0,blend_radius_m)
    |   movel([0.130924, -1.336621, -2.596664, -0.779104, 1.570796, 1.701720],accel_mss,speed_ms,0,blend_radius_m)
    |   movel([0.133454, -1.336091, -2.597007, -0.779292, 1.570796, 1.704250],accel_mss,speed_ms,0,blend_radius_m)
    |   movel([0.135896, -1.335925, -2.597114, -0.779351, 1.570796, 1.706692],accel_mss,speed_ms,0,blend_radius_m)
    |   movel([0.138205, -1.336142, -2.596974, -0.779274, 1.570796, 1.709002],accel_mss,speed_ms,0,blend_radius_m)
    |   movel([0.140282, -1.336752, -2.596579, -0.779057, 1.570796, 1.711078],accel_mss,speed_ms,0,blend_radius_m)
    |   movel([0.142032, -1.337718, -2.595955, -0.778716, 1.570796, 1.712829],accel_mss,speed_ms,0,blend_radius_m)
    |   movel([0.143439, -1.339008, -2.595118, -0.778262, 1.570796, 1.714235],accel_mss,speed_ms,0,blend_radius_m)
    |   movel([0.144488, -1.340588, -2.594091, -0.777710, 1.570796, 1.715284],accel_mss,speed_ms,0,blend_radius_m)
    |   movel([0.145165, -1.342423, -2.592894, -0.777072, 1.570796, 1.715961],accel_mss,speed_ms,0,blend_radius_m)
    |   movel([0.145455, -1.344478, -2.591547, -0.776364, 1.570796, 1.716251],accel_mss,speed_ms,0,blend_radius_m)
    |   movel([0.145344, -1.346722, -2.590071, -0.775597, 1.570796, 1.716141],accel_mss,speed_ms,0,blend_radius_m)
    |   movel([0.144824, -1.349115, -2.588487, -0.774786, 1.570796, 1.715620],accel_mss,speed_ms,0,blend_radius_m)
    |   movel([0.144168, -1.350936, -2.587278, -0.774175, 1.570796, 1.714964],accel_mss,speed_ms,0,blend_radius_m)
    |   movel([0.143799, -1.351553, -2.586867, -0.773969, 1.570796, 1.714595],accel_mss,speed_ms,0,blend_radius_m)
    |   movel([0.143353, -1.352016, -2.586559, -0.773815, 1.570796, 1.714149],accel_mss,speed_ms,0,blend_radius_m)
    |   movel([0.142793, -1.352352, -2.586334, -0.773703, 1.570796, 1.713589],accel_mss,speed_ms,0,blend_radius_m)
    |   movel([0.142084, -1.352591, -2.586175, -0.773623, 1.570796, 1.712880],accel_mss,speed_ms,0,blend_radius_m)
    |   movel([0.140076, -1.352892, -2.585973, -0.773523, 1.570796, 1.710872],accel_mss,speed_ms,0,blend_radius_m)
    |   movel([0.140788, -1.349617, -2.588155, -0.774617, 1.570796, 1.711585],accel_mss,speed_ms,0,blend_radius_m)
    |   movel([0.141097, -1.346826, -2.590002, -0.775561, 1.570796, 1.711893],accel_mss,speed_ms,0,blend_radius_m)
    |   movel([0.140994, -1.344508, -2.591528, -0.776354, 1.570796, 1.711790],accel_mss,speed_ms,0,blend_radius_m)
    |   movel([0.140462, -1.342652, -2.592744, -0.776993, 1.570796, 1.711258],accel_mss,speed_ms,0,blend_radius_m)
    |   movel([0.140033, -1.341891, -2.593241, -0.777256, 1.570796, 1.710829],accel_mss,speed_ms,0,blend_radius_m)
    |   movel([0.139494, -1.341240, -2.593666, -0.777483, 1.570796, 1.710290],accel_mss,speed_ms,0,blend_radius_m)
    |   movel([0.138842, -1.340698, -2.594020, -0.777671, 1.570796, 1.709638],accel_mss,speed_ms,0,blend_radius_m)
    |   movel([0.137202, -1.339931, -2.594519, -0.777939, 1.570796, 1.707998],accel_mss,speed_ms,0,blend_radius_m)
    |   movel([0.136209, -1.339702, -2.594668, -0.778019, 1.570796, 1.707005],accel_mss,speed_ms,0,blend_radius_m)
    |   movel([0.133874, -1.339543, -2.594771, -0.778075, 1.570796, 1.704670],accel_mss,speed_ms,0,blend_radius_m)
    |   movel([0.131737, -1.339758, -2.594631, -0.778000, 1.570796, 1.702534],accel_mss,speed_ms,0,blend_radius_m)
    |   movel([0.129547, -1.340326, -2.594262, -0.777801, 1.570796, 1.700343],accel_mss,speed_ms,0,blend_radius_m)
    |   movel([0.127354, -1.341213, -2.593684, -0.777492, 1.570796, 1.698150],accel_mss,speed_ms,0,blend_radius_m)
    |   movel([0.125210, -1.342385, -2.592919, -0.777086, 1.570796, 1.696007],accel_mss,speed_ms,0,blend_radius_m)
    |   movel([0.123173, -1.343809, -2.591986, -0.776594, 1.570796, 1.693969],accel_mss,speed_ms,0,blend_radius_m)
    |   movel([0.121287, -1.345453, -2.590906, -0.776030, 1.570796, 1.692083],accel_mss,speed_ms,0,blend_radius_m)
    |   movel([0.119605, -1.347280, -2.589702, -0.775407, 1.570796, 1.690401],accel_mss,speed_ms,0,blend_radius_m)
    |   movel([0.118176, -1.349262, -2.588390, -0.774737, 1.570796, 1.688972],accel_mss,speed_ms,0,blend_radius_m)
    |   movel([0.116876, -1.351632, -2.586814, -0.773942, 1.570796, 1.687673],accel_mss,speed_ms,0,blend_radius_m)
    |   movel([0.116086, -1.353795, -2.585370, -0.773224, 1.570796, 1.686883],accel_mss,speed_ms,0,blend_radius_m)
    |   movel([0.115884, -1.354803, -2.584694, -0.772892, 1.570796, 1.686680],accel_mss,speed_ms,0,blend_radius_m)
    |   movel([0.115866, -1.356690, -2.583426, -0.772273, 1.570796, 1.686662],accel_mss,speed_ms,0,blend_radius_m)
    |   movel([0.116049, -1.357571, -2.582832, -0.771986, 1.570796, 1.686846],accel_mss,speed_ms,0,blend_radius_m)
    |   movel([0.116806, -1.359220, -2.581717, -0.771452, 1.570796, 1.687602],accel_mss,speed_ms,0,blend_radius_m)
    |   movel([0.118084, -1.360738, -2.580688, -0.770963, 1.570796, 1.688880],accel_mss,speed_ms,0,blend_radius_m)
    |   movel([0.119883, -1.362140, -2.579735, -0.770515, 1.570796, 1.690680],accel_mss,speed_ms,0,blend_radius_m)
    |   movel([0.122207, -1.363446, -2.578844, -0.770099, 1.570796, 1.693003],accel_mss,speed_ms,0,blend_radius_m)
    |   movel([0.120970, -1.365764, -2.577257, -0.769368, 1.570796, 1.691767],accel_mss,speed_ms,0,blend_radius_m)
    |   speed_ms = 0.005
    |   # Splitting Linear movement in 4 (instruction 644: MoveL 596)
    |   movel([0.120970, -1.363576, -2.576244, -0.772569, 1.570796, 1.691767],accel_mss,speed_ms,0,blend_radius_m)
    |   movel([0.120970, -1.361399, -2.575227, -0.775763, 1.570796, 1.691767],accel_mss,speed_ms,0,blend_radius_m)
    |   movel([0.120970, -1.359233, -2.574206, -0.778950, 1.570796, 1.691767],accel_mss,speed_ms,0,blend_radius_m)
    |   movel([0.120970, -1.357076, -2.573181, -0.782131, 1.570796, 1.691767],accel_mss,speed_ms,0,blend_radius_m)
    |   speed_ms = 0.040
    |   # Splitting Linear movement in 18 (instruction 646: MoveL 597)
    |   movel([0.120281, -1.355463, -2.574272, -0.782653, 1.570796, 1.691078],accel_mss,speed_ms,0,blend_radius_m)
    |   movel([0.119589, -1.353848, -2.575361, -0.783180, 1.570796, 1.690386],accel_mss,speed_ms,0,blend_radius_m)
    |   movel([0.118894, -1.352231, -2.576448, -0.783711, 1.570796, 1.689691],accel_mss,speed_ms,0,blend_radius_m)
    |   movel([0.118196, -1.350611, -2.577532, -0.784246, 1.570796, 1.688993],accel_mss,speed_ms,0,blend_radius_m)
    |   movel([0.117496, -1.348989, -2.578614, -0.784786, 1.570796, 1.688292],accel_mss,speed_ms,0,blend_radius_m)
    |   movel([0.116792, -1.347365, -2.579694, -0.785330, 1.570796, 1.687588],accel_mss,speed_ms,0,blend_radius_m)
    |   movel([0.116085, -1.345739, -2.580772, -0.785878, 1.570796, 1.686882],accel_mss,speed_ms,0,blend_radius_m)
    |   movel([0.115376, -1.344111, -2.581848, -0.786430, 1.570796, 1.686172],accel_mss,speed_ms,0,blend_radius_m)
    |   movel([0.114663, -1.342481, -2.582921, -0.786987, 1.570796, 1.685460],accel_mss,speed_ms,0,blend_radius_m)
    |   movel([0.113948, -1.340849, -2.583992, -0.787548, 1.570796, 1.684744],accel_mss,speed_ms,0,blend_radius_m)
    |   movel([0.113229, -1.339214, -2.585061, -0.788114, 1.570796, 1.684025],accel_mss,speed_ms,0,blend_radius_m)
    |   movel([0.112508, -1.337577, -2.586128, -0.788684, 1.570796, 1.683304],accel_mss,speed_ms,0,blend_radius_m)
    |   movel([0.111783, -1.335939, -2.587193, -0.789258, 1.570796, 1.682579],accel_mss,speed_ms,0,blend_radius_m)
    |   movel([0.111055, -1.334298, -2.588255, -0.789836, 1.570796, 1.681852],accel_mss,speed_ms,0,blend_radius_m)
    |   movel([0.110324, -1.332654, -2.589315, -0.790419, 1.570796, 1.681121],accel_mss,speed_ms,0,blend_radius_m)
    |   movel([0.109590, -1.331009, -2.590373, -0.791007, 1.570796, 1.680387],accel_mss,speed_ms,0,blend_radius_m)
    |   movel([0.108853, -1.329362, -2.591428, -0.791599, 1.570796, 1.679650],accel_mss,speed_ms,0,blend_radius_m)
    |   movel([0.108113, -1.327712, -2.592482, -0.792195, 1.570796, 1.678910],accel_mss,speed_ms,0,blend_radius_m)
    |   speed_ms = 0.005
    |   # Splitting Linear movement in 4 (instruction 648: MoveL 598)
    |   movel([0.108113, -1.329914, -2.593538, -0.788936, 1.570796, 1.678910],accel_mss,speed_ms,0,blend_radius_m)
    |   movel([0.108113, -1.332127, -2.594591, -0.785670, 1.570796, 1.678910],accel_mss,speed_ms,0,blend_radius_m)
    |   movel([0.108113, -1.334352, -2.595641, -0.782397, 1.570796, 1.678910],accel_mss,speed_ms,0,blend_radius_m)
    |   movel([0.108113, -1.336587, -2.596686, -0.779116, 1.570796, 1.678910],accel_mss,speed_ms,0,blend_radius_m)
    |   speed_ms = 0.035
    |   movel([0.106316, -1.338548, -2.595417, -0.778424, 1.570796, 1.677112],accel_mss,speed_ms,0,blend_radius_m)
    |   movel([0.104661, -1.340518, -2.594137, -0.777734, 1.570796, 1.675458],accel_mss,speed_ms,0,blend_radius_m)
    |   movel([0.103151, -1.342493, -2.592848, -0.777048, 1.570796, 1.673947],accel_mss,speed_ms,0,blend_radius_m)
    |   movel([0.101779, -1.344469, -2.591553, -0.776367, 1.570796, 1.672575],accel_mss,speed_ms,0,blend_radius_m)
    |   movel([0.100547, -1.346438, -2.590257, -0.775693, 1.570796, 1.671344],accel_mss,speed_ms,0,blend_radius_m)
    |   movel([0.099454, -1.348400, -2.588962, -0.775028, 1.570796, 1.670250],accel_mss,speed_ms,0,blend_radius_m)
    |   movel([0.098494, -1.350345, -2.587671, -0.774373, 1.570796, 1.669290],accel_mss,speed_ms,0,blend_radius_m)
    |   movel([0.097668, -1.352272, -2.586388, -0.773729, 1.570796, 1.668464],accel_mss,speed_ms,0,blend_radius_m)
    |   movel([0.096975, -1.354174, -2.585116, -0.773099, 1.570796, 1.667771],accel_mss,speed_ms,0,blend_radius_m)
    |   movel([0.096414, -1.356048, -2.583858, -0.772483, 1.570796, 1.667210],accel_mss,speed_ms,0,blend_radius_m)
    |   movel([0.095669, -1.359690, -2.581399, -0.771300, 1.570796, 1.666466],accel_mss,speed_ms,0,blend_radius_m)
    |   movel([0.095485, -1.361452, -2.580203, -0.770734, 1.570796, 1.666281],accel_mss,speed_ms,0,blend_radius_m)
    |   movel([0.095485, -1.364830, -2.577897, -0.769662, 1.570796, 1.666281],accel_mss,speed_ms,0,blend_radius_m)
    |   movel([0.095663, -1.366440, -2.576793, -0.769156, 1.570796, 1.666459],accel_mss,speed_ms,0,blend_radius_m)
    |   movel([0.096371, -1.369483, -2.574695, -0.768211, 1.570796, 1.667167],accel_mss,speed_ms,0,blend_radius_m)
    |   movel([0.096895, -1.370908, -2.573708, -0.767773, 1.570796, 1.667692],accel_mss,speed_ms,0,blend_radius_m)
    |   movel([0.098286, -1.373539, -2.571879, -0.766971, 1.570796, 1.669082],accel_mss,speed_ms,0,blend_radius_m)
    |   movel([0.099145, -1.374741, -2.571040, -0.766608, 1.570796, 1.669941],accel_mss,speed_ms,0,blend_radius_m)
    |   movel([0.101187, -1.376891, -2.569534, -0.765964, 1.570796, 1.671984],accel_mss,speed_ms,0,blend_radius_m)
    |   movel([0.102370, -1.377834, -2.568871, -0.765684, 1.570796, 1.673166],accel_mss,speed_ms,0,blend_radius_m)
    |   movel([0.103656, -1.378683, -2.568274, -0.765432, 1.570796, 1.674453],accel_mss,speed_ms,0,blend_radius_m)
    |   movel([0.105046, -1.379436, -2.567743, -0.765210, 1.570796, 1.675842],accel_mss,speed_ms,0,blend_radius_m)
    |   movel([0.106539, -1.380083, -2.567286, -0.765020, 1.570796, 1.677335],accel_mss,speed_ms,0,blend_radius_m)
    |   movel([0.108133, -1.380628, -2.566901, -0.764860, 1.570796, 1.678929],accel_mss,speed_ms,0,blend_radius_m)
    |   movel([0.109829, -1.381061, -2.566595, -0.764734, 1.570796, 1.680626],accel_mss,speed_ms,0,blend_radius_m)
    |   movel([0.111627, -1.381379, -2.566369, -0.764641, 1.570796, 1.682423],accel_mss,speed_ms,0,blend_radius_m)
    |   movel([0.113523, -1.381580, -2.566227, -0.764582, 1.570796, 1.684320],accel_mss,speed_ms,0,blend_radius_m)
    |   movel([0.112735, -1.383387, -2.564944, -0.764058, 1.570796, 1.683531],accel_mss,speed_ms,0,blend_radius_m)
    |   movel([0.112369, -1.384047, -2.564474, -0.763868, 1.570796, 1.683166],accel_mss,speed_ms,0,blend_radius_m)
    |   movel([0.111916, -1.384464, -2.564177, -0.763748, 1.570796, 1.682713],accel_mss,speed_ms,0,blend_radius_m)
    |   movel([0.111348, -1.384668, -2.564032, -0.763689, 1.570796, 1.682144],accel_mss,speed_ms,0,blend_radius_m)
    |   movel([0.110638, -1.384685, -2.564020, -0.763685, 1.570796, 1.681434],accel_mss,speed_ms,0,blend_radius_m)
    |   movel([0.107947, -1.384329, -2.564273, -0.763787, 1.570796, 1.678743],accel_mss,speed_ms,0,blend_radius_m)
    |   movel([0.105434, -1.383717, -2.564709, -0.763963, 1.570796, 1.676230],accel_mss,speed_ms,0,blend_radius_m)
    |   movel([0.103104, -1.382861, -2.565318, -0.764210, 1.570796, 1.673901],accel_mss,speed_ms,0,blend_radius_m)
    |   movel([0.100967, -1.381773, -2.566090, -0.764526, 1.570796, 1.671763],accel_mss,speed_ms,0,blend_radius_m)
    |   movel([0.099025, -1.380467, -2.567014, -0.764907, 1.570796, 1.669822],accel_mss,speed_ms,0,blend_radius_m)
    |   movel([0.097291, -1.378954, -2.568083, -0.765352, 1.570796, 1.668087],accel_mss,speed_ms,0,blend_radius_m)
    |   movel([0.095771, -1.377246, -2.569285, -0.765858, 1.570796, 1.666568],accel_mss,speed_ms,0,blend_radius_m)
    |   movel([0.094473, -1.375356, -2.570610, -0.766423, 1.570796, 1.665270],accel_mss,speed_ms,0,blend_radius_m)
    |   movel([0.093411, -1.373293, -2.572051, -0.767046, 1.570796, 1.664208],accel_mss,speed_ms,0,blend_radius_m)
    |   movel([0.092590, -1.371070, -2.573596, -0.767723, 1.570796, 1.663386],accel_mss,speed_ms,0,blend_radius_m)
    |   movel([0.092021, -1.368697, -2.575238, -0.768454, 1.570796, 1.662818],accel_mss,speed_ms,0,blend_radius_m)
    |   movel([0.091719, -1.366186, -2.576967, -0.769236, 1.570796, 1.662515],accel_mss,speed_ms,0,blend_radius_m)
    |   movel([0.091688, -1.363552, -2.578771, -0.770066, 1.570796, 1.662485],accel_mss,speed_ms,0,blend_radius_m)
    |   movel([0.091943, -1.360805, -2.580642, -0.770941, 1.570796, 1.662739],accel_mss,speed_ms,0,blend_radius_m)
    |   movel([0.092496, -1.357956, -2.582572, -0.771861, 1.570796, 1.663292],accel_mss,speed_ms,0,blend_radius_m)
    |   movel([0.093354, -1.355018, -2.584550, -0.772821, 1.570796, 1.664150],accel_mss,speed_ms,0,blend_radius_m)
    |   movel([0.095047, -1.350740, -2.587409, -0.774241, 1.570796, 1.665843],accel_mss,speed_ms,0,blend_radius_m)
    |   movel([0.096067, -1.348618, -2.588817, -0.774954, 1.570796, 1.666864],accel_mss,speed_ms,0,blend_radius_m)
    |   movel([0.097206, -1.346508, -2.590212, -0.775670, 1.570796, 1.668002],accel_mss,speed_ms,0,blend_radius_m)
    |   movel([0.098471, -1.344407, -2.591594, -0.776388, 1.570796, 1.669267],accel_mss,speed_ms,0,blend_radius_m)
    |   movel([0.099865, -1.342317, -2.592963, -0.777109, 1.570796, 1.670662],accel_mss,speed_ms,0,blend_radius_m)
    |   movel([0.101395, -1.340234, -2.594321, -0.777833, 1.570796, 1.672192],accel_mss,speed_ms,0,blend_radius_m)
    |   movel([0.103062, -1.338162, -2.595667, -0.778560, 1.570796, 1.673858],accel_mss,speed_ms,0,blend_radius_m)
    |   movel([0.104534, -1.336491, -2.596748, -0.779150, 1.570796, 1.675330],accel_mss,speed_ms,0,blend_radius_m)
    |   movel([0.105082, -1.336014, -2.597056, -0.779319, 1.570796, 1.675878],accel_mss,speed_ms,0,blend_radius_m)
    |   movel([0.105579, -1.335755, -2.597223, -0.779411, 1.570796, 1.676375],accel_mss,speed_ms,0,blend_radius_m)
    |   movel([0.106077, -1.335699, -2.597259, -0.779431, 1.570796, 1.676873],accel_mss,speed_ms,0,blend_radius_m)
    |   movel([0.106628, -1.335829, -2.597175, -0.779385, 1.570796, 1.677424],accel_mss,speed_ms,0,blend_radius_m)
    |   movel([0.108113, -1.336587, -2.596686, -0.779116, 1.570796, 1.678910],accel_mss,speed_ms,0,blend_radius_m)
    |   movel([0.106316, -1.338548, -2.595417, -0.778424, 1.570796, 1.677112],accel_mss,speed_ms,0,blend_radius_m)
    |   movel([0.106109, -1.338793, -2.595258, -0.778338, 1.570796, 1.676906],accel_mss,speed_ms,0,blend_radius_m)
    |   speed_ms = 0.005
    |   # Splitting Linear movement in 6 (instruction 714: MoveL 662)
    |   movel([0.106109, -1.337304, -2.594563, -0.780522, 1.570796, 1.676906],accel_mss,speed_ms,0,blend_radius_m)
    |   movel([0.106109, -1.335819, -2.593867, -0.782703, 1.570796, 1.676906],accel_mss,speed_ms,0,blend_radius_m)
    |   movel([0.106109, -1.334340, -2.593168, -0.784880, 1.570796, 1.676906],accel_mss,speed_ms,0,blend_radius_m)
    |   movel([0.106109, -1.332866, -2.592468, -0.787055, 1.570796, 1.676906],accel_mss,speed_ms,0,blend_radius_m)
    |   movel([0.106109, -1.331396, -2.591767, -0.789226, 1.570796, 1.676906],accel_mss,speed_ms,0,blend_radius_m)
    |   movel([0.106109, -1.329932, -2.591064, -0.791393, 1.570796, 1.676906],accel_mss,speed_ms,0,blend_radius_m)
    |   speed_ms = 0.040
    |   # Splitting Linear movement in 20 (instruction 716: MoveL 663)
    |   movel([0.106875, -1.327668, -2.592510, -0.792211, 1.570796, 1.677671],accel_mss,speed_ms,0,blend_radius_m)
    |   movel([0.107644, -1.325396, -2.593955, -0.793038, 1.570796, 1.678441],accel_mss,speed_ms,0,blend_radius_m)
    |   movel([0.108418, -1.323116, -2.595398, -0.793875, 1.570796, 1.679214],accel_mss,speed_ms,0,blend_radius_m)
    |   movel([0.109195, -1.320828, -2.596839, -0.794722, 1.570796, 1.679991],accel_mss,speed_ms,0,blend_radius_m)
    |   movel([0.109976, -1.318531, -2.598279, -0.795579, 1.570796, 1.680773],accel_mss,speed_ms,0,blend_radius_m)
    |   movel([0.110761, -1.316226, -2.599717, -0.796446, 1.570796, 1.681558],accel_mss,speed_ms,0,blend_radius_m)
    |   movel([0.111551, -1.313912, -2.601153, -0.797324, 1.570796, 1.682347],accel_mss,speed_ms,0,blend_radius_m)
    |   movel([0.112344, -1.311590, -2.602588, -0.798212, 1.570796, 1.683140],accel_mss,speed_ms,0,blend_radius_m)
    |   movel([0.113141, -1.309259, -2.604021, -0.799110, 1.570796, 1.683938],accel_mss,speed_ms,0,blend_radius_m)
    |   movel([0.113943, -1.306919, -2.605452, -0.800018, 1.570796, 1.684739],accel_mss,speed_ms,0,blend_radius_m)
    |   movel([0.114748, -1.304570, -2.606881, -0.800938, 1.570796, 1.685545],accel_mss,speed_ms,0,blend_radius_m)
    |   movel([0.115558, -1.302212, -2.608309, -0.801867, 1.570796, 1.686354],accel_mss,speed_ms,0,blend_radius_m)
    |   movel([0.116372, -1.299846, -2.609735, -0.802808, 1.570796, 1.687168],accel_mss,speed_ms,0,blend_radius_m)
    |   movel([0.117190, -1.297470, -2.611159, -0.803759, 1.570796, 1.687987],accel_mss,speed_ms,0,blend_radius_m)
    |   movel([0.118013, -1.295086, -2.612582, -0.804722, 1.570796, 1.688809],accel_mss,speed_ms,0,blend_radius_m)
    |   movel([0.118839, -1.292692, -2.614002, -0.805695, 1.570796, 1.689636],accel_mss,speed_ms,0,blend_radius_m)
    |   movel([0.119671, -1.290288, -2.615421, -0.806679, 1.570796, 1.690467],accel_mss,speed_ms,0,blend_radius_m)
    |   movel([0.120506, -1.287876, -2.616838, -0.807675, 1.570796, 1.691302],accel_mss,speed_ms,0,blend_radius_m)
    |   movel([0.121346, -1.285454, -2.618253, -0.808682, 1.570796, 1.692142],accel_mss,speed_ms,0,blend_radius_m)
    |   movel([0.122190, -1.283022, -2.619667, -0.809700, 1.570796, 1.692987],accel_mss,speed_ms,0,blend_radius_m)
    |   speed_ms = 0.005
    |   # Splitting Linear movement in 6 (instruction 718: MoveL 664)
    |   movel([0.122190, -1.284530, -2.620405, -0.807454, 1.570796, 1.692987],accel_mss,speed_ms,0,blend_radius_m)
    |   movel([0.122190, -1.286044, -2.621141, -0.805204, 1.570796, 1.692987],accel_mss,speed_ms,0,blend_radius_m)
    |   movel([0.122190, -1.287564, -2.621876, -0.802950, 1.570796, 1.692987],accel_mss,speed_ms,0,blend_radius_m)
    |   movel([0.122190, -1.289088, -2.622609, -0.800692, 1.570796, 1.692987],accel_mss,speed_ms,0,blend_radius_m)
    |   movel([0.122190, -1.290619, -2.623340, -0.798430, 1.570796, 1.692987],accel_mss,speed_ms,0,blend_radius_m)
    |   movel([0.122190, -1.292154, -2.624070, -0.796165, 1.570796, 1.692987],accel_mss,speed_ms,0,blend_radius_m)
    |   speed_ms = 0.035
    |   movel([0.121345, -1.294131, -2.622907, -0.795351, 1.570796, 1.692142],accel_mss,speed_ms,0,blend_radius_m)
    |   movel([0.120728, -1.295999, -2.621802, -0.794587, 1.570796, 1.691524],accel_mss,speed_ms,0,blend_radius_m)
    |   movel([0.120340, -1.297760, -2.620758, -0.793872, 1.570796, 1.691137],accel_mss,speed_ms,0,blend_radius_m)
    |   movel([0.120177, -1.299417, -2.619771, -0.793202, 1.570796, 1.690973],accel_mss,speed_ms,0,blend_radius_m)
    |   movel([0.120238, -1.300972, -2.618841, -0.792576, 1.570796, 1.691034],accel_mss,speed_ms,0,blend_radius_m)
    |   movel([0.120525, -1.302426, -2.617969, -0.791994, 1.570796, 1.691322],accel_mss,speed_ms,0,blend_radius_m)
    |   movel([0.121039, -1.303782, -2.617154, -0.791453, 1.570796, 1.691835],accel_mss,speed_ms,0,blend_radius_m)
    |   movel([0.121775, -1.305043, -2.616393, -0.790953, 1.570796, 1.692571],accel_mss,speed_ms,0,blend_radius_m)
    |   movel([0.123160, -1.306558, -2.615477, -0.790354, 1.570796, 1.693956],accel_mss,speed_ms,0,blend_radius_m)
    |   movel([0.124887, -1.307667, -2.614804, -0.789918, 1.570796, 1.695683],accel_mss,speed_ms,0,blend_radius_m)
    |   movel([0.126906, -1.308379, -2.614372, -0.789639, 1.570796, 1.697702],accel_mss,speed_ms,0,blend_radius_m)
    |   movel([0.129165, -1.308691, -2.614181, -0.789516, 1.570796, 1.699961],accel_mss,speed_ms,0,blend_radius_m)
    |   movel([0.131624, -1.308604, -2.614234, -0.789550, 1.570796, 1.702420],accel_mss,speed_ms,0,blend_radius_m)
    |   movel([0.134231, -1.308122, -2.614527, -0.789739, 1.570796, 1.705027],accel_mss,speed_ms,0,blend_radius_m)
    |   movel([0.136947, -1.307240, -2.615063, -0.790086, 1.570796, 1.707743],accel_mss,speed_ms,0,blend_radius_m)
    |   movel([0.139721, -1.305954, -2.615843, -0.790593, 1.570796, 1.710517],accel_mss,speed_ms,0,blend_radius_m)
    |   movel([0.142427, -1.304314, -2.616833, -0.791242, 1.570796, 1.713223],accel_mss,speed_ms,0,blend_radius_m)
    |   movel([0.144947, -1.302401, -2.617985, -0.792004, 1.570796, 1.715744],accel_mss,speed_ms,0,blend_radius_m)
    |   movel([0.147248, -1.300261, -2.619267, -0.792861, 1.570796, 1.718044],accel_mss,speed_ms,0,blend_radius_m)
    |   movel([0.149284, -1.297939, -2.620651, -0.793799, 1.570796, 1.720081],accel_mss,speed_ms,0,blend_radius_m)
    |   movel([0.151023, -1.295483, -2.622108, -0.794798, 1.570796, 1.721819],accel_mss,speed_ms,0,blend_radius_m)
    |   movel([0.152413, -1.292947, -2.623604, -0.795838, 1.570796, 1.723209],accel_mss,speed_ms,0,blend_radius_m)
    |   movel([0.153421, -1.290374, -2.625114, -0.796901, 1.570796, 1.724218],accel_mss,speed_ms,0,blend_radius_m)
    |   movel([0.153997, -1.287818, -2.626605, -0.797966, 1.570796, 1.724793],accel_mss,speed_ms,0,blend_radius_m)
    |   movel([0.154134, -1.285249, -2.628096, -0.799045, 1.570796, 1.724930],accel_mss,speed_ms,0,blend_radius_m)
    |   movel([0.153815, -1.282956, -2.629419, -0.800014, 1.570796, 1.724612],accel_mss,speed_ms,0,blend_radius_m)
    |   movel([0.153057, -1.280974, -2.630557, -0.800858, 1.570796, 1.723854],accel_mss,speed_ms,0,blend_radius_m)
    |   movel([0.151885, -1.279327, -2.631500, -0.801562, 1.570796, 1.722682],accel_mss,speed_ms,0,blend_radius_m)
    |   movel([0.150315, -1.278045, -2.632231, -0.802113, 1.570796, 1.721111],accel_mss,speed_ms,0,blend_radius_m)
    |   movel([0.148371, -1.277155, -2.632737, -0.802497, 1.570796, 1.719168],accel_mss,speed_ms,0,blend_radius_m)
    |   movel([0.146077, -1.276685, -2.633004, -0.802699, 1.570796, 1.716873],accel_mss,speed_ms,0,blend_radius_m)
    |   movel([0.143454, -1.276662, -2.633017, -0.802710, 1.570796, 1.714250],accel_mss,speed_ms,0,blend_radius_m)
    |   movel([0.141686, -1.276947, -2.632856, -0.802586, 1.570796, 1.712483],accel_mss,speed_ms,0,blend_radius_m)
    |   movel([0.141035, -1.277197, -2.632713, -0.802478, 1.570796, 1.711832],accel_mss,speed_ms,0,blend_radius_m)
    |   movel([0.140530, -1.277531, -2.632524, -0.802335, 1.570796, 1.711326],accel_mss,speed_ms,0,blend_radius_m)
    |   movel([0.140166, -1.277948, -2.632286, -0.802155, 1.570796, 1.710962],accel_mss,speed_ms,0,blend_radius_m)
    |   movel([0.139936, -1.278464, -2.631992, -0.801933, 1.570796, 1.710733],accel_mss,speed_ms,0,blend_radius_m)
    |   movel([0.139857, -1.279803, -2.631228, -0.801358, 1.570796, 1.710654],accel_mss,speed_ms,0,blend_radius_m)
    |   movel([0.140062, -1.280163, -2.631022, -0.801204, 1.570796, 1.710859],accel_mss,speed_ms,0,blend_radius_m)
    |   movel([0.140512, -1.280424, -2.630872, -0.801092, 1.570796, 1.711308],accel_mss,speed_ms,0,blend_radius_m)
    |   movel([0.141094, -1.280569, -2.630790, -0.801031, 1.570796, 1.711890],accel_mss,speed_ms,0,blend_radius_m)
    |   movel([0.143913, -1.280620, -2.630760, -0.801009, 1.570796, 1.714709],accel_mss,speed_ms,0,blend_radius_m)
    |   movel([0.145854, -1.281094, -2.630488, -0.800806, 1.570796, 1.716650],accel_mss,speed_ms,0,blend_radius_m)
    |   movel([0.147474, -1.281968, -2.629987, -0.800434, 1.570796, 1.718271],accel_mss,speed_ms,0,blend_radius_m)
    |   movel([0.148747, -1.283195, -2.629281, -0.799913, 1.570796, 1.719543],accel_mss,speed_ms,0,blend_radius_m)
    |   movel([0.149631, -1.284731, -2.628395, -0.799263, 1.570796, 1.720427],accel_mss,speed_ms,0,blend_radius_m)
    |   movel([0.150095, -1.286531, -2.627353, -0.798505, 1.570796, 1.720892],accel_mss,speed_ms,0,blend_radius_m)
    |   movel([0.150108, -1.288549, -2.626179, -0.797661, 1.570796, 1.720905],accel_mss,speed_ms,0,blend_radius_m)
    |   movel([0.149938, -1.289625, -2.625552, -0.797212, 1.570796, 1.720734],accel_mss,speed_ms,0,blend_radius_m)
    |   movel([0.149201, -1.291951, -2.624189, -0.796249, 1.570796, 1.719997],accel_mss,speed_ms,0,blend_radius_m)
    |   movel([0.148659, -1.293144, -2.623488, -0.795757, 1.570796, 1.719455],accel_mss,speed_ms,0,blend_radius_m)
    |   movel([0.147296, -1.295452, -2.622126, -0.794811, 1.570796, 1.718093],accel_mss,speed_ms,0,blend_radius_m)
    |   movel([0.145613, -1.297615, -2.620844, -0.793930, 1.570796, 1.716410],accel_mss,speed_ms,0,blend_radius_m)
    |   movel([0.143668, -1.299586, -2.619670, -0.793133, 1.570796, 1.714464],accel_mss,speed_ms,0,blend_radius_m)
    |   movel([0.141512, -1.301317, -2.618635, -0.792437, 1.570796, 1.712308],accel_mss,speed_ms,0,blend_radius_m)
    |   movel([0.139201, -1.302763, -2.617767, -0.791859, 1.570796, 1.709997],accel_mss,speed_ms,0,blend_radius_m)
    |   movel([0.136788, -1.303874, -2.617098, -0.791417, 1.570796, 1.707584],accel_mss,speed_ms,0,blend_radius_m)
    |   movel([0.135561, -1.304290, -2.616847, -0.791251, 1.570796, 1.706357],accel_mss,speed_ms,0,blend_radius_m)
    |   movel([0.134326, -1.304607, -2.616656, -0.791125, 1.570796, 1.705123],accel_mss,speed_ms,0,blend_radius_m)
    |   movel([0.131994, -1.304898, -2.616481, -0.791010, 1.570796, 1.702791],accel_mss,speed_ms,0,blend_radius_m)
    |   movel([0.129883, -1.304757, -2.616566, -0.791066, 1.570796, 1.700680],accel_mss,speed_ms,0,blend_radius_m)
    |   movel([0.128042, -1.304210, -2.616896, -0.791283, 1.570796, 1.698839],accel_mss,speed_ms,0,blend_radius_m)
    |   movel([0.126514, -1.303287, -2.617452, -0.791650, 1.570796, 1.697310],accel_mss,speed_ms,0,blend_radius_m)
    |   movel([0.125344, -1.302019, -2.618213, -0.792156, 1.570796, 1.696140],accel_mss,speed_ms,0,blend_radius_m)
    |   movel([0.124583, -1.300429, -2.619166, -0.792794, 1.570796, 1.695379],accel_mss,speed_ms,0,blend_radius_m)
    |   movel([0.124369, -1.299522, -2.619708, -0.793159, 1.570796, 1.695165],accel_mss,speed_ms,0,blend_radius_m)
    |   movel([0.124274, -1.298549, -2.620288, -0.793552, 1.570796, 1.695070],accel_mss,speed_ms,0,blend_radius_m)
    |   movel([0.124471, -1.296400, -2.621565, -0.794424, 1.570796, 1.695267],accel_mss,speed_ms,0,blend_radius_m)
    |   movel([0.124610, -1.294832, -2.622493, -0.795064, 1.570796, 1.695406],accel_mss,speed_ms,0,blend_radius_m)
    |   movel([0.124287, -1.293651, -2.623190, -0.795549, 1.570796, 1.695083],accel_mss,speed_ms,0,blend_radius_m)
    |   movel([0.123483, -1.292783, -2.623701, -0.795906, 1.570796, 1.694280],accel_mss,speed_ms,0,blend_radius_m)
    |   movel([0.122190, -1.292154, -2.624070, -0.796165, 1.570796, 1.692987],accel_mss,speed_ms,0,blend_radius_m)
    |   movel([0.121345, -1.294131, -2.622907, -0.795351, 1.570796, 1.692142],accel_mss,speed_ms,0,blend_radius_m)
    |   movel([0.121138, -1.294760, -2.622535, -0.795094, 1.570796, 1.691935],accel_mss,speed_ms,0,blend_radius_m)
    |   speed_ms = 0.005
    |   # Splitting Linear movement in 4 (instruction 795: MoveL 739)
    |   movel([0.121138, -1.292462, -2.621443, -0.798484, 1.570796, 1.691935],accel_mss,speed_ms,0,blend_radius_m)
    |   movel([0.121138, -1.290176, -2.620347, -0.801866, 1.570796, 1.691935],accel_mss,speed_ms,0,blend_radius_m)
    |   movel([0.121138, -1.287903, -2.619247, -0.805239, 1.570796, 1.691935],accel_mss,speed_ms,0,blend_radius_m)
    |   movel([0.121138, -1.285642, -2.618144, -0.808603, 1.570796, 1.691935],accel_mss,speed_ms,0,blend_radius_m)
    |   speed_ms = 0.040
    |   # Splitting Linear movement in 10 (instruction 797: MoveL 740)
    |   movel([0.120168, -1.283891, -2.619163, -0.809336, 1.570796, 1.690965],accel_mss,speed_ms,0,blend_radius_m)
    |   movel([0.119193, -1.282138, -2.620179, -0.810072, 1.570796, 1.689990],accel_mss,speed_ms,0,blend_radius_m)
    |   movel([0.118214, -1.280383, -2.621192, -0.810813, 1.570796, 1.689011],accel_mss,speed_ms,0,blend_radius_m)
    |   movel([0.117231, -1.278627, -2.622202, -0.811559, 1.570796, 1.688027],accel_mss,speed_ms,0,blend_radius_m)
    |   movel([0.116242, -1.276870, -2.623210, -0.812310, 1.570796, 1.687039],accel_mss,speed_ms,0,blend_radius_m)
    |   movel([0.115250, -1.275110, -2.624214, -0.813064, 1.570796, 1.686046],accel_mss,speed_ms,0,blend_radius_m)
    |   movel([0.114252, -1.273349, -2.625216, -0.813824, 1.570796, 1.685049],accel_mss,speed_ms,0,blend_radius_m)
    |   movel([0.113250, -1.271587, -2.626215, -0.814588, 1.570796, 1.684047],accel_mss,speed_ms,0,blend_radius_m)
    |   movel([0.112244, -1.269823, -2.627210, -0.815356, 1.570796, 1.683040],accel_mss,speed_ms,0,blend_radius_m)
    |   movel([0.111232, -1.268057, -2.628203, -0.816129, 1.570796, 1.682029],accel_mss,speed_ms,0,blend_radius_m)
    |   speed_ms = 0.005
    |   # Splitting Linear movement in 6 (instruction 799: MoveL 741)
    |   movel([0.111232, -1.269578, -2.628952, -0.813859, 1.570796, 1.682029],accel_mss,speed_ms,0,blend_radius_m)
    |   movel([0.111232, -1.271104, -2.629700, -0.811585, 1.570796, 1.682029],accel_mss,speed_ms,0,blend_radius_m)
    |   movel([0.111232, -1.272636, -2.630446, -0.809307, 1.570796, 1.682029],accel_mss,speed_ms,0,blend_radius_m)
    |   movel([0.111232, -1.274174, -2.631190, -0.807025, 1.570796, 1.682029],accel_mss,speed_ms,0,blend_radius_m)
    |   movel([0.111232, -1.275718, -2.631933, -0.804739, 1.570796, 1.682029],accel_mss,speed_ms,0,blend_radius_m)
    |   movel([0.111232, -1.277267, -2.632674, -0.802448, 1.570796, 1.682029],accel_mss,speed_ms,0,blend_radius_m)
    |   speed_ms = 0.035
    |   movel([0.108593, -1.280168, -2.631019, -0.801202, 1.570796, 1.679389],accel_mss,speed_ms,0,blend_radius_m)
    |   movel([0.106209, -1.283173, -2.629294, -0.799922, 1.570796, 1.677005],accel_mss,speed_ms,0,blend_radius_m)
    |   movel([0.104085, -1.286253, -2.627514, -0.798622, 1.570796, 1.674882],accel_mss,speed_ms,0,blend_radius_m)
    |   movel([0.102227, -1.289384, -2.625692, -0.797313, 1.570796, 1.673023],accel_mss,speed_ms,0,blend_radius_m)
    |   movel([0.100631, -1.292543, -2.623841, -0.796004, 1.570796, 1.671427],accel_mss,speed_ms,0,blend_radius_m)
    |   movel([0.099307, -1.295700, -2.621979, -0.794709, 1.570796, 1.670103],accel_mss,speed_ms,0,blend_radius_m)
    |   movel([0.098254, -1.298838, -2.620116, -0.793435, 1.570796, 1.669050],accel_mss,speed_ms,0,blend_radius_m)
    |   movel([0.097473, -1.301928, -2.618268, -0.792193, 1.570796, 1.668269],accel_mss,speed_ms,0,blend_radius_m)
    |   movel([0.096969, -1.304953, -2.616448, -0.790988, 1.570796, 1.667765],accel_mss,speed_ms,0,blend_radius_m)
    |   movel([0.096738, -1.307891, -2.614668, -0.789830, 1.570796, 1.667534],accel_mss,speed_ms,0,blend_radius_m)
    |   movel([0.096788, -1.310719, -2.612945, -0.788726, 1.570796, 1.667584],accel_mss,speed_ms,0,blend_radius_m)
    |   movel([0.097117, -1.313419, -2.611289, -0.787681, 1.570796, 1.667913],accel_mss,speed_ms,0,blend_radius_m)
    |   movel([0.097729, -1.315967, -2.609718, -0.786704, 1.570796, 1.668525],accel_mss,speed_ms,0,blend_radius_m)
    |   movel([0.098624, -1.318345, -2.608244, -0.785800, 1.570796, 1.669421],accel_mss,speed_ms,0,blend_radius_m)
    |   movel([0.099806, -1.320537, -2.606879, -0.784973, 1.570796, 1.670603],accel_mss,speed_ms,0,blend_radius_m)
    |   movel([0.101278, -1.322521, -2.605637, -0.784231, 1.570796, 1.672074],accel_mss,speed_ms,0,blend_radius_m)
    |   movel([0.103099, -1.324348, -2.604490, -0.783551, 1.570796, 1.673895],accel_mss,speed_ms,0,blend_radius_m)
    |   movel([0.105155, -1.325898, -2.603512, -0.782978, 1.570796, 1.675952],accel_mss,speed_ms,0,blend_radius_m)
    |   movel([0.107423, -1.327177, -2.602704, -0.782508, 1.570796, 1.678219],accel_mss,speed_ms,0,blend_radius_m)
    |   movel([0.109886, -1.328189, -2.602063, -0.782138, 1.570796, 1.680682],accel_mss,speed_ms,0,blend_radius_m)
    |   movel([0.112523, -1.328935, -2.601588, -0.781865, 1.570796, 1.683319],accel_mss,speed_ms,0,blend_radius_m)
    |   movel([0.115317, -1.329419, -2.601281, -0.781689, 1.570796, 1.686113],accel_mss,speed_ms,0,blend_radius_m)
    |   movel([0.118243, -1.329644, -2.601138, -0.781607, 1.570796, 1.689040],accel_mss,speed_ms,0,blend_radius_m)
    |   movel([0.121288, -1.329611, -2.601158, -0.781619, 1.570796, 1.692084],accel_mss,speed_ms,0,blend_radius_m)
    |   movel([0.124434, -1.329319, -2.601344, -0.781725, 1.570796, 1.695230],accel_mss,speed_ms,0,blend_radius_m)
    |   movel([0.127659, -1.328771, -2.601693, -0.781925, 1.570796, 1.698455],accel_mss,speed_ms,0,blend_radius_m)
    |   movel([0.130948, -1.327968, -2.602202, -0.782218, 1.570796, 1.701744],accel_mss,speed_ms,0,blend_radius_m)
    |   movel([0.134283, -1.326904, -2.602876, -0.782608, 1.570796, 1.705080],accel_mss,speed_ms,0,blend_radius_m)
    |   movel([0.137648, -1.325584, -2.603711, -0.783094, 1.570796, 1.708444],accel_mss,speed_ms,0,blend_radius_m)
    |   movel([0.141024, -1.324002, -2.604707, -0.783680, 1.570796, 1.711820],accel_mss,speed_ms,0,blend_radius_m)
    |   movel([0.144395, -1.322155, -2.605866, -0.784367, 1.570796, 1.715191],accel_mss,speed_ms,0,blend_radius_m)
    |   movel([0.147741, -1.320044, -2.607186, -0.785159, 1.570796, 1.718537],accel_mss,speed_ms,0,blend_radius_m)
    |   movel([0.151168, -1.317594, -2.608710, -0.786085, 1.570796, 1.721964],accel_mss,speed_ms,0,blend_radius_m)
    |   movel([0.154411, -1.314986, -2.610324, -0.787079, 1.570796, 1.725207],accel_mss,speed_ms,0,blend_radius_m)
    |   movel([0.157467, -1.312239, -2.612014, -0.788137, 1.570796, 1.728264],accel_mss,speed_ms,0,blend_radius_m)
    |   movel([0.160325, -1.309362, -2.613773, -0.789254, 1.570796, 1.731121],accel_mss,speed_ms,0,blend_radius_m)
    |   movel([0.162972, -1.306375, -2.615588, -0.790426, 1.570796, 1.733769],accel_mss,speed_ms,0,blend_radius_m)
    |   movel([0.165403, -1.303289, -2.617450, -0.791649, 1.570796, 1.736199],accel_mss,speed_ms,0,blend_radius_m)
    |   movel([0.167601, -1.300122, -2.619350, -0.792917, 1.570796, 1.738397],accel_mss,speed_ms,0,blend_radius_m)
    |   movel([0.169559, -1.296891, -2.621274, -0.794225, 1.570796, 1.740356],accel_mss,speed_ms,0,blend_radius_m)
    |   movel([0.171264, -1.293612, -2.623212, -0.795564, 1.570796, 1.742060],accel_mss,speed_ms,0,blend_radius_m)
    |   movel([0.172702, -1.290301, -2.625157, -0.796932, 1.570796, 1.743498],accel_mss,speed_ms,0,blend_radius_m)
    |   movel([0.173861, -1.286980, -2.627092, -0.798317, 1.570796, 1.744657],accel_mss,speed_ms,0,blend_radius_m)
    |   movel([0.174729, -1.283664, -2.629011, -0.799714, 1.570796, 1.745525],accel_mss,speed_ms,0,blend_radius_m)
    |   movel([0.175291, -1.280373, -2.630902, -0.801114, 1.570796, 1.746087],accel_mss,speed_ms,0,blend_radius_m)
    |   movel([0.175532, -1.277129, -2.632752, -0.802508, 1.570796, 1.746328],accel_mss,speed_ms,0,blend_radius_m)
    |   movel([0.175444, -1.273952, -2.634551, -0.803885, 1.570796, 1.746240],accel_mss,speed_ms,0,blend_radius_m)
    |   movel([0.175005, -1.270864, -2.636289, -0.805236, 1.570796, 1.745801],accel_mss,speed_ms,0,blend_radius_m)
    |   movel([0.174329, -1.268363, -2.637687, -0.806339, 1.570796, 1.745126],accel_mss,speed_ms,0,blend_radius_m)
    |   movel([0.173383, -1.266072, -2.638961, -0.807356, 1.570796, 1.744180],accel_mss,speed_ms,0,blend_radius_m)
    |   movel([0.172181, -1.264000, -2.640108, -0.808281, 1.570796, 1.742977],accel_mss,speed_ms,0,blend_radius_m)
    |   movel([0.170744, -1.262142, -2.641132, -0.809115, 1.570796, 1.741540],accel_mss,speed_ms,0,blend_radius_m)
    |   movel([0.169097, -1.260502, -2.642032, -0.809855, 1.570796, 1.739893],accel_mss,speed_ms,0,blend_radius_m)
    |   movel([0.167259, -1.259083, -2.642808, -0.810498, 1.570796, 1.738056],accel_mss,speed_ms,0,blend_radius_m)
    |   movel([0.165253, -1.257886, -2.643461, -0.811042, 1.570796, 1.736049],accel_mss,speed_ms,0,blend_radius_m)
    |   movel([0.163103, -1.256911, -2.643991, -0.811486, 1.570796, 1.733899],accel_mss,speed_ms,0,blend_radius_m)
    |   movel([0.160832, -1.256154, -2.644403, -0.811832, 1.570796, 1.731628],accel_mss,speed_ms,0,blend_radius_m)
    |   movel([0.158462, -1.255622, -2.644691, -0.812076, 1.570796, 1.729259],accel_mss,speed_ms,0,blend_radius_m)
    |   movel([0.156018, -1.255309, -2.644861, -0.812219, 1.570796, 1.726815],accel_mss,speed_ms,0,blend_radius_m)
    |   movel([0.153526, -1.255212, -2.644913, -0.812264, 1.570796, 1.724323],accel_mss,speed_ms,0,blend_radius_m)
    |   movel([0.151007, -1.255333, -2.644848, -0.812208, 1.570796, 1.721803],accel_mss,speed_ms,0,blend_radius_m)
    |   movel([0.148489, -1.255670, -2.644665, -0.812054, 1.570796, 1.719285],accel_mss,speed_ms,0,blend_radius_m)
    |   movel([0.145992, -1.256215, -2.644370, -0.811805, 1.570796, 1.716788],accel_mss,speed_ms,0,blend_radius_m)
    |   movel([0.143542, -1.256970, -2.643959, -0.811459, 1.570796, 1.714338],accel_mss,speed_ms,0,blend_radius_m)
    |   movel([0.142953, -1.258946, -2.642883, -0.810560, 1.570796, 1.713750],accel_mss,speed_ms,0,blend_radius_m)
    |   movel([0.142872, -1.259553, -2.642551, -0.810285, 1.570796, 1.713668],accel_mss,speed_ms,0,blend_radius_m)
    |   movel([0.142954, -1.259947, -2.642336, -0.810106, 1.570796, 1.713750],accel_mss,speed_ms,0,blend_radius_m)
    |   movel([0.143214, -1.260161, -2.642218, -0.810009, 1.570796, 1.714011],accel_mss,speed_ms,0,blend_radius_m)
    |   movel([0.143675, -1.260219, -2.642187, -0.809983, 1.570796, 1.714472],accel_mss,speed_ms,0,blend_radius_m)
    |   movel([0.148316, -1.259566, -2.642544, -0.810279, 1.570796, 1.719112],accel_mss,speed_ms,0,blend_radius_m)
    |   movel([0.151240, -1.259402, -2.642634, -0.810353, 1.570796, 1.722037],accel_mss,speed_ms,0,blend_radius_m)
    |   movel([0.154010, -1.259502, -2.642579, -0.810308, 1.570796, 1.724806],accel_mss,speed_ms,0,blend_radius_m)
    |   movel([0.156618, -1.259862, -2.642382, -0.810145, 1.570796, 1.727415],accel_mss,speed_ms,0,blend_radius_m)
    |   movel([0.159047, -1.260471, -2.642049, -0.809869, 1.570796, 1.729843],accel_mss,speed_ms,0,blend_radius_m)
    |   movel([0.161290, -1.261319, -2.641584, -0.809486, 1.570796, 1.732086],accel_mss,speed_ms,0,blend_radius_m)
    |   movel([0.163333, -1.262398, -2.640991, -0.809000, 1.570796, 1.734129],accel_mss,speed_ms,0,blend_radius_m)
    |   movel([0.165170, -1.263699, -2.640274, -0.808416, 1.570796, 1.735967],accel_mss,speed_ms,0,blend_radius_m)
    |   movel([0.166792, -1.265208, -2.639440, -0.807741, 1.570796, 1.737588],accel_mss,speed_ms,0,blend_radius_m)
    |   movel([0.168184, -1.266921, -2.638489, -0.806978, 1.570796, 1.738981],accel_mss,speed_ms,0,blend_radius_m)
    |   movel([0.169340, -1.268822, -2.637431, -0.806136, 1.570796, 1.740137],accel_mss,speed_ms,0,blend_radius_m)
    |   movel([0.170255, -1.270903, -2.636267, -0.805219, 1.570796, 1.741051],accel_mss,speed_ms,0,blend_radius_m)
    |   movel([0.170920, -1.273150, -2.635004, -0.804235, 1.570796, 1.741716],accel_mss,speed_ms,0,blend_radius_m)
    |   movel([0.171322, -1.275556, -2.633644, -0.803188, 1.570796, 1.742118],accel_mss,speed_ms,0,blend_radius_m)
    |   movel([0.171458, -1.278110, -2.632194, -0.802085, 1.570796, 1.742254],accel_mss,speed_ms,0,blend_radius_m)
    |   movel([0.171323, -1.280801, -2.630657, -0.800931, 1.570796, 1.742119],accel_mss,speed_ms,0,blend_radius_m)
    |   movel([0.170903, -1.283674, -2.629005, -0.799710, 1.570796, 1.741699],accel_mss,speed_ms,0,blend_radius_m)
    |   movel([0.170233, -1.286556, -2.627338, -0.798495, 1.570796, 1.741029],accel_mss,speed_ms,0,blend_radius_m)
    |   movel([0.169320, -1.289436, -2.625662, -0.797291, 1.570796, 1.740116],accel_mss,speed_ms,0,blend_radius_m)
    |   movel([0.168181, -1.292297, -2.623986, -0.796106, 1.570796, 1.738977],accel_mss,speed_ms,0,blend_radius_m)
    |   movel([0.166826, -1.295128, -2.622318, -0.794943, 1.570796, 1.737623],accel_mss,speed_ms,0,blend_radius_m)
    |   movel([0.165266, -1.297912, -2.620667, -0.793810, 1.570796, 1.736062],accel_mss,speed_ms,0,blend_radius_m)
    |   movel([0.163518, -1.300639, -2.619041, -0.792710, 1.570796, 1.734314],accel_mss,speed_ms,0,blend_radius_m)
    |   movel([0.161587, -1.303295, -2.617447, -0.791647, 1.570796, 1.732383],accel_mss,speed_ms,0,blend_radius_m)
    |   movel([0.159488, -1.305867, -2.615895, -0.790627, 1.570796, 1.730285],accel_mss,speed_ms,0,blend_radius_m)
    |   movel([0.157233, -1.308347, -2.614391, -0.789651, 1.570796, 1.728029],accel_mss,speed_ms,0,blend_radius_m)
    |   movel([0.154830, -1.310722, -2.612942, -0.788724, 1.570796, 1.725626],accel_mss,speed_ms,0,blend_radius_m)
    |   movel([0.152288, -1.312978, -2.611560, -0.787851, 1.570796, 1.723084],accel_mss,speed_ms,0,blend_radius_m)
    |   movel([0.149618, -1.315105, -2.610250, -0.787034, 1.570796, 1.720415],accel_mss,speed_ms,0,blend_radius_m)
    |   movel([0.146830, -1.317095, -2.609019, -0.786274, 1.570796, 1.717627],accel_mss,speed_ms,0,blend_radius_m)
    |   movel([0.143935, -1.318936, -2.607877, -0.785577, 1.570796, 1.714732],accel_mss,speed_ms,0,blend_radius_m)
    |   movel([0.140937, -1.320613, -2.606831, -0.784945, 1.570796, 1.711733],accel_mss,speed_ms,0,blend_radius_m)
    |   movel([0.138227, -1.321940, -2.606001, -0.784447, 1.570796, 1.709024],accel_mss,speed_ms,0,blend_radius_m)
    |   movel([0.135534, -1.323081, -2.605286, -0.784022, 1.570796, 1.706330],accel_mss,speed_ms,0,blend_radius_m)
    |   movel([0.132865, -1.324033, -2.604688, -0.783668, 1.570796, 1.703661],accel_mss,speed_ms,0,blend_radius_m)
    |   movel([0.130234, -1.324801, -2.604204, -0.783383, 1.570796, 1.701030],accel_mss,speed_ms,0,blend_radius_m)
    |   movel([0.127647, -1.325385, -2.603836, -0.783168, 1.570796, 1.698443],accel_mss,speed_ms,0,blend_radius_m)
    |   movel([0.125117, -1.325788, -2.603582, -0.783019, 1.570796, 1.695913],accel_mss,speed_ms,0,blend_radius_m)
    |   movel([0.122651, -1.326005, -2.603445, -0.782939, 1.570796, 1.693448],accel_mss,speed_ms,0,blend_radius_m)
    |   movel([0.120258, -1.326044, -2.603420, -0.782925, 1.570796, 1.691054],accel_mss,speed_ms,0,blend_radius_m)
    |   movel([0.117950, -1.325902, -2.603510, -0.782977, 1.570796, 1.688747],accel_mss,speed_ms,0,blend_radius_m)
    |   movel([0.115738, -1.325579, -2.603714, -0.783096, 1.570796, 1.686534],accel_mss,speed_ms,0,blend_radius_m)
    |   movel([0.113627, -1.325076, -2.604031, -0.783282, 1.570796, 1.684424],accel_mss,speed_ms,0,blend_radius_m)
    |   movel([0.111633, -1.324391, -2.604463, -0.783536, 1.570796, 1.682430],accel_mss,speed_ms,0,blend_radius_m)
    |   movel([0.109765, -1.323523, -2.605009, -0.783858, 1.570796, 1.680561],accel_mss,speed_ms,0,blend_radius_m)
    |   movel([0.108035, -1.322471, -2.605669, -0.784249, 1.570796, 1.678831],accel_mss,speed_ms,0,blend_radius_m)
    |   movel([0.106450, -1.321237, -2.606441, -0.784711, 1.570796, 1.677246],accel_mss,speed_ms,0,blend_radius_m)
    |   movel([0.105024, -1.319816, -2.607328, -0.785245, 1.570796, 1.675820],accel_mss,speed_ms,0,blend_radius_m)
    |   movel([0.103789, -1.318233, -2.608313, -0.785842, 1.570796, 1.674585],accel_mss,speed_ms,0,blend_radius_m)
    |   movel([0.102760, -1.316511, -2.609381, -0.786497, 1.570796, 1.673556],accel_mss,speed_ms,0,blend_radius_m)
    |   movel([0.101937, -1.314662, -2.610523, -0.787203, 1.570796, 1.672734],accel_mss,speed_ms,0,blend_radius_m)
    |   movel([0.101320, -1.312692, -2.611735, -0.787961, 1.570796, 1.672116],accel_mss,speed_ms,0,blend_radius_m)
    |   movel([0.100909, -1.310613, -2.613009, -0.788767, 1.570796, 1.671706],accel_mss,speed_ms,0,blend_radius_m)
    |   movel([0.100706, -1.308435, -2.614337, -0.789617, 1.570796, 1.671503],accel_mss,speed_ms,0,blend_radius_m)
    |   movel([0.100706, -1.306167, -2.615714, -0.790509, 1.570796, 1.671502],accel_mss,speed_ms,0,blend_radius_m)
    |   movel([0.100914, -1.303816, -2.617134, -0.791440, 1.570796, 1.671710],accel_mss,speed_ms,0,blend_radius_m)
    |   movel([0.101330, -1.301397, -2.618587, -0.792405, 1.570796, 1.672126],accel_mss,speed_ms,0,blend_radius_m)
    |   movel([0.101950, -1.298919, -2.620068, -0.793403, 1.570796, 1.672746],accel_mss,speed_ms,0,blend_radius_m)
    |   movel([0.102777, -1.296391, -2.621570, -0.794428, 1.570796, 1.673573],accel_mss,speed_ms,0,blend_radius_m)
    |   movel([0.103813, -1.293823, -2.623088, -0.795478, 1.570796, 1.674610],accel_mss,speed_ms,0,blend_radius_m)
    |   movel([0.105054, -1.291232, -2.624611, -0.796546, 1.570796, 1.675850],accel_mss,speed_ms,0,blend_radius_m)
    |   movel([0.106503, -1.288625, -2.626135, -0.797629, 1.570796, 1.677299],accel_mss,speed_ms,0,blend_radius_m)
    |   movel([0.108159, -1.286013, -2.627653, -0.798723, 1.570796, 1.678955],accel_mss,speed_ms,0,blend_radius_m)
    |   movel([0.110023, -1.283411, -2.629157, -0.799821, 1.570796, 1.680819],accel_mss,speed_ms,0,blend_radius_m)
    |   movel([0.113606, -1.278818, -2.631790, -0.801781, 1.570796, 1.684402],accel_mss,speed_ms,0,blend_radius_m)
    |   movel([0.112390, -1.277888, -2.632320, -0.802181, 1.570796, 1.683186],accel_mss,speed_ms,0,blend_radius_m)
    |   movel([0.111232, -1.277267, -2.632674, -0.802448, 1.570796, 1.682029],accel_mss,speed_ms,0,blend_radius_m)
    |   movel([0.109028, -1.279691, -2.631292, -0.801406, 1.570796, 1.679824],accel_mss,speed_ms,0,blend_radius_m)
    |   speed_ms = 0.005
    |   # Splitting Linear movement in 6 (instruction 939: MoveL 879)
    |   movel([0.109028, -1.278144, -2.630553, -0.803693, 1.570796, 1.679824],accel_mss,speed_ms,0,blend_radius_m)
    |   movel([0.109028, -1.276602, -2.629812, -0.805975, 1.570796, 1.679824],accel_mss,speed_ms,0,blend_radius_m)
    |   movel([0.109028, -1.275067, -2.629069, -0.808253, 1.570796, 1.679824],accel_mss,speed_ms,0,blend_radius_m)
    |   movel([0.109028, -1.273537, -2.628325, -0.810527, 1.570796, 1.679824],accel_mss,speed_ms,0,blend_radius_m)
    |   movel([0.109028, -1.272012, -2.627580, -0.812797, 1.570796, 1.679824],accel_mss,speed_ms,0,blend_radius_m)
    |   movel([0.109028, -1.270493, -2.626832, -0.815063, 1.570796, 1.679824],accel_mss,speed_ms,0,blend_radius_m)
    |   speed_ms = 0.040
    |   # Splitting Linear movement in 24 (instruction 941: MoveL 880)
    |   movel([0.111193, -1.268211, -2.628117, -0.816061, 1.570796, 1.681990],accel_mss,speed_ms,0,blend_radius_m)
    |   movel([0.113368, -1.265921, -2.629399, -0.817069, 1.570796, 1.684164],accel_mss,speed_ms,0,blend_radius_m)
    |   movel([0.115552, -1.263624, -2.630679, -0.818086, 1.570796, 1.686348],accel_mss,speed_ms,0,blend_radius_m)
    |   movel([0.117745, -1.261320, -2.631956, -0.819113, 1.570796, 1.688542],accel_mss,speed_ms,0,blend_radius_m)
    |   movel([0.119948, -1.259008, -2.633232, -0.820150, 1.570796, 1.690744],accel_mss,speed_ms,0,blend_radius_m)
    |   movel([0.122160, -1.256689, -2.634504, -0.821196, 1.570796, 1.692957],accel_mss,speed_ms,0,blend_radius_m)
    |   movel([0.124382, -1.254362, -2.635775, -0.822252, 1.570796, 1.695179],accel_mss,speed_ms,0,blend_radius_m)
    |   movel([0.126614, -1.252028, -2.637043, -0.823318, 1.570796, 1.697410],accel_mss,speed_ms,0,blend_radius_m)
    |   movel([0.128855, -1.249686, -2.638308, -0.824395, 1.570796, 1.699651],accel_mss,speed_ms,0,blend_radius_m)
    |   movel([0.131106, -1.247337, -2.639571, -0.825481, 1.570796, 1.701902],accel_mss,speed_ms,0,blend_radius_m)
    |   movel([0.133367, -1.244980, -2.640832, -0.826577, 1.570796, 1.704163],accel_mss,speed_ms,0,blend_radius_m)
    |   movel([0.135637, -1.242615, -2.642090, -0.827684, 1.570796, 1.706433],accel_mss,speed_ms,0,blend_radius_m)
    |   movel([0.137917, -1.240243, -2.643346, -0.828801, 1.570796, 1.708714],accel_mss,speed_ms,0,blend_radius_m)
    |   movel([0.140208, -1.237863, -2.644599, -0.829928, 1.570796, 1.711004],accel_mss,speed_ms,0,blend_radius_m)
    |   movel([0.142508, -1.235475, -2.645849, -0.831065, 1.570796, 1.713304],accel_mss,speed_ms,0,blend_radius_m)
    |   movel([0.144818, -1.233079, -2.647097, -0.832213, 1.570796, 1.715615],accel_mss,speed_ms,0,blend_radius_m)
    |   movel([0.147139, -1.230675, -2.648343, -0.833371, 1.570796, 1.717935],accel_mss,speed_ms,0,blend_radius_m)
    |   movel([0.149470, -1.228263, -2.649586, -0.834540, 1.570796, 1.720266],accel_mss,speed_ms,0,blend_radius_m)
    |   movel([0.151811, -1.225843, -2.650826, -0.835719, 1.570796, 1.722607],accel_mss,speed_ms,0,blend_radius_m)
    |   movel([0.154162, -1.223416, -2.652064, -0.836909, 1.570796, 1.724958],accel_mss,speed_ms,0,blend_radius_m)
    |   movel([0.156523, -1.220980, -2.653299, -0.838110, 1.570796, 1.727320],accel_mss,speed_ms,0,blend_radius_m)
    |   movel([0.158895, -1.218535, -2.654532, -0.839322, 1.570796, 1.729692],accel_mss,speed_ms,0,blend_radius_m)
    |   movel([0.161278, -1.216083, -2.655762, -0.840544, 1.570796, 1.732074],accel_mss,speed_ms,0,blend_radius_m)
    |   movel([0.163671, -1.213622, -2.656989, -0.841778, 1.570796, 1.734467],accel_mss,speed_ms,0,blend_radius_m)
    |   speed_ms = 0.005
    |   # Splitting Linear movement in 6 (instruction 943: MoveL 881)
    |   movel([0.163671, -1.215182, -2.657779, -0.839429, 1.570796, 1.734467],accel_mss,speed_ms,0,blend_radius_m)
    |   movel([0.163671, -1.216747, -2.658567, -0.837075, 1.570796, 1.734467],accel_mss,speed_ms,0,blend_radius_m)
    |   movel([0.163671, -1.218320, -2.659354, -0.834716, 1.570796, 1.734467],accel_mss,speed_ms,0,blend_radius_m)
    |   movel([0.163671, -1.219898, -2.660139, -0.832352, 1.570796, 1.734467],accel_mss,speed_ms,0,blend_radius_m)
    |   movel([0.163671, -1.221484, -2.660922, -0.829983, 1.570796, 1.734467],accel_mss,speed_ms,0,blend_radius_m)
    |   movel([0.163671, -1.223075, -2.661704, -0.827609, 1.570796, 1.734467],accel_mss,speed_ms,0,blend_radius_m)
    |   speed_ms = 0.035
    |   movel([0.165524, -1.220284, -2.663106, -0.828999, 1.570796, 1.736320],accel_mss,speed_ms,0,blend_radius_m)
    |   movel([0.166959, -1.217407, -2.664542, -0.830440, 1.570796, 1.737756],accel_mss,speed_ms,0,blend_radius_m)
    |   movel([0.167968, -1.214511, -2.665977, -0.831901, 1.570796, 1.738764],accel_mss,speed_ms,0,blend_radius_m)
    |   movel([0.168538, -1.211673, -2.667375, -0.833341, 1.570796, 1.739335],accel_mss,speed_ms,0,blend_radius_m)
    |   movel([0.168667, -1.208964, -2.668700, -0.834724, 1.570796, 1.739464],accel_mss,speed_ms,0,blend_radius_m)
    |   movel([0.168338, -1.206464, -2.669917, -0.836008, 1.570796, 1.739135],accel_mss,speed_ms,0,blend_radius_m)
    |   movel([0.167542, -1.204247, -2.670989, -0.837152, 1.570796, 1.738339],accel_mss,speed_ms,0,blend_radius_m)
    |   movel([0.166271, -1.202398, -2.671880, -0.838111, 1.570796, 1.737068],accel_mss,speed_ms,0,blend_radius_m)
    |   movel([0.165405, -1.201580, -2.672272, -0.838536, 1.570796, 1.736201],accel_mss,speed_ms,0,blend_radius_m)
    |   movel([0.164430, -1.200891, -2.672603, -0.838895, 1.570796, 1.735227],accel_mss,speed_ms,0,blend_radius_m)
    |   movel([0.162198, -1.199899, -2.673077, -0.839412, 1.570796, 1.732994],accel_mss,speed_ms,0,blend_radius_m)
    |   movel([0.159641, -1.199420, -2.673306, -0.839663, 1.570796, 1.730437],accel_mss,speed_ms,0,blend_radius_m)
    |   movel([0.156820, -1.199452, -2.673291, -0.839646, 1.570796, 1.727616],accel_mss,speed_ms,0,blend_radius_m)
    |   movel([0.153804, -1.199984, -2.673037, -0.839368, 1.570796, 1.724600],accel_mss,speed_ms,0,blend_radius_m)
    |   movel([0.150659, -1.201012, -2.672545, -0.838832, 1.570796, 1.721455],accel_mss,speed_ms,0,blend_radius_m)
    |   movel([0.147454, -1.202526, -2.671818, -0.838045, 1.570796, 1.718250],accel_mss,speed_ms,0,blend_radius_m)
    |   movel([0.144260, -1.204511, -2.670862, -0.837016, 1.570796, 1.715057],accel_mss,speed_ms,0,blend_radius_m)
    |   movel([0.141097, -1.206964, -2.669674, -0.835751, 1.570796, 1.711893],accel_mss,speed_ms,0,blend_radius_m)
    |   movel([0.138253, -1.209644, -2.668368, -0.834376, 1.570796, 1.709050],accel_mss,speed_ms,0,blend_radius_m)
    |   movel([0.135764, -1.212500, -2.666968, -0.832920, 1.570796, 1.706560],accel_mss,speed_ms,0,blend_radius_m)
    |   movel([0.133664, -1.215470, -2.665503, -0.831416, 1.570796, 1.704460],accel_mss,speed_ms,0,blend_radius_m)
    |   movel([0.131980, -1.218499, -2.663998, -0.829892, 1.570796, 1.702776],accel_mss,speed_ms,0,blend_radius_m)
    |   movel([0.130744, -1.221539, -2.662477, -0.828373, 1.570796, 1.701540],accel_mss,speed_ms,0,blend_radius_m)
    |   movel([0.129983, -1.224537, -2.660967, -0.826885, 1.570796, 1.700779],accel_mss,speed_ms,0,blend_radius_m)
    |   movel([0.129724, -1.227446, -2.659492, -0.825452, 1.570796, 1.700520],accel_mss,speed_ms,0,blend_radius_m)
    |   movel([0.129934, -1.229675, -2.658354, -0.824359, 1.570796, 1.700730],accel_mss,speed_ms,0,blend_radius_m)
    |   movel([0.130525, -1.231703, -2.657315, -0.823371, 1.570796, 1.701322],accel_mss,speed_ms,0,blend_radius_m)
    |   movel([0.131450, -1.233479, -2.656401, -0.822509, 1.570796, 1.702247],accel_mss,speed_ms,0,blend_radius_m)
    |   movel([0.132666, -1.234963, -2.655634, -0.821792, 1.570796, 1.703462],accel_mss,speed_ms,0,blend_radius_m)
    |   movel([0.134124, -1.236113, -2.655038, -0.821238, 1.570796, 1.704920],accel_mss,speed_ms,0,blend_radius_m)
    |   movel([0.135782, -1.236881, -2.654639, -0.820869, 1.570796, 1.706578],accel_mss,speed_ms,0,blend_radius_m)
    |   movel([0.137600, -1.237226, -2.654460, -0.820703, 1.570796, 1.708396],accel_mss,speed_ms,0,blend_radius_m)
    |   movel([0.138555, -1.237225, -2.654461, -0.820704, 1.570796, 1.709352],accel_mss,speed_ms,0,blend_radius_m)
    |   movel([0.139535, -1.237098, -2.654527, -0.820764, 1.570796, 1.710332],accel_mss,speed_ms,0,blend_radius_m)
    |   movel([0.141303, -1.233679, -2.656298, -0.822412, 1.570796, 1.712099],accel_mss,speed_ms,0,blend_radius_m)
    |   movel([0.138607, -1.232270, -2.657023, -0.823095, 1.570796, 1.709403],accel_mss,speed_ms,0,blend_radius_m)
    |   movel([0.136534, -1.230664, -2.657848, -0.823877, 1.570796, 1.707330],accel_mss,speed_ms,0,blend_radius_m)
    |   movel([0.135733, -1.229782, -2.658300, -0.824307, 1.570796, 1.706529],accel_mss,speed_ms,0,blend_radius_m)
    |   movel([0.134591, -1.227857, -2.659282, -0.825250, 1.570796, 1.705387],accel_mss,speed_ms,0,blend_radius_m)
    |   movel([0.134255, -1.226810, -2.659815, -0.825764, 1.570796, 1.705052],accel_mss,speed_ms,0,blend_radius_m)
    |   movel([0.134077, -1.225703, -2.660376, -0.826309, 1.570796, 1.704874],accel_mss,speed_ms,0,blend_radius_m)
    |   movel([0.134054, -1.224540, -2.660965, -0.826884, 1.570796, 1.704851],accel_mss,speed_ms,0,blend_radius_m)
    |   movel([0.134191, -1.223313, -2.661584, -0.827491, 1.570796, 1.704987],accel_mss,speed_ms,0,blend_radius_m)
    |   movel([0.134481, -1.222028, -2.662232, -0.828130, 1.570796, 1.705277],accel_mss,speed_ms,0,blend_radius_m)
    |   movel([0.134932, -1.220674, -2.662911, -0.828804, 1.570796, 1.705729],accel_mss,speed_ms,0,blend_radius_m)
    |   movel([0.135539, -1.219261, -2.663618, -0.829510, 1.570796, 1.706335],accel_mss,speed_ms,0,blend_radius_m)
    |   movel([0.137231, -1.216231, -2.665126, -0.831032, 1.570796, 1.708028],accel_mss,speed_ms,0,blend_radius_m)
    |   movel([0.139152, -1.213569, -2.666442, -0.832378, 1.570796, 1.709948],accel_mss,speed_ms,0,blend_radius_m)
    |   movel([0.141361, -1.211137, -2.667638, -0.833614, 1.570796, 1.712157],accel_mss,speed_ms,0,blend_radius_m)
    |   movel([0.143791, -1.208983, -2.668691, -0.834715, 1.570796, 1.714588],accel_mss,speed_ms,0,blend_radius_m)
    |   movel([0.146381, -1.207147, -2.669585, -0.835657, 1.570796, 1.717177],accel_mss,speed_ms,0,blend_radius_m)
    |   movel([0.149060, -1.205677, -2.670298, -0.836414, 1.570796, 1.719857],accel_mss,speed_ms,0,blend_radius_m)
    |   movel([0.151762, -1.204617, -2.670811, -0.836961, 1.570796, 1.722558],accel_mss,speed_ms,0,blend_radius_m)
    |   movel([0.154417, -1.204010, -2.671104, -0.837275, 1.570796, 1.725214],accel_mss,speed_ms,0,blend_radius_m)
    |   movel([0.156959, -1.203898, -2.671158, -0.837333, 1.570796, 1.727755],accel_mss,speed_ms,0,blend_radius_m)
    |   movel([0.158199, -1.204043, -2.671088, -0.837258, 1.570796, 1.728995],accel_mss,speed_ms,0,blend_radius_m)
    |   movel([0.160342, -1.204717, -2.670762, -0.836909, 1.570796, 1.731138],accel_mss,speed_ms,0,blend_radius_m)
    |   movel([0.161243, -1.205245, -2.670507, -0.836637, 1.570796, 1.732040],accel_mss,speed_ms,0,blend_radius_m)
    |   movel([0.162708, -1.206664, -2.669820, -0.835905, 1.570796, 1.733504],accel_mss,speed_ms,0,blend_radius_m)
    |   movel([0.163720, -1.208559, -2.668898, -0.834932, 1.570796, 1.734517],accel_mss,speed_ms,0,blend_radius_m)
    |   movel([0.164122, -1.210040, -2.668175, -0.834174, 1.570796, 1.734919],accel_mss,speed_ms,0,blend_radius_m)
    |   movel([0.164273, -1.211595, -2.667413, -0.833381, 1.570796, 1.735070],accel_mss,speed_ms,0,blend_radius_m)
    |   movel([0.164184, -1.213218, -2.666615, -0.832556, 1.570796, 1.734981],accel_mss,speed_ms,0,blend_radius_m)
    |   movel([0.163871, -1.214904, -2.665783, -0.831702, 1.570796, 1.734667],accel_mss,speed_ms,0,blend_radius_m)
    |   movel([0.163341, -1.216647, -2.664919, -0.830823, 1.570796, 1.734138],accel_mss,speed_ms,0,blend_radius_m)
